// TwinCAT 3 PLC project Struckig
// Title: Struckig
// Company: Stefan Besler
// Author: Stefan Besler and contributers
// ProjectVersion: 0.19.4.0
// Description: Full port of pantor ruckig library (Community version) to IEC 61131-3 Structured Text. Online Trajectory Generation. Real-time. Time-optimal. Jerk-constrained.
// ProgramVersion: 3.1.4026.18
// project tree:
//   / Constants.TcGVL, ParameterList.TcGVL
//   Struckig/Block/ BlockInterval.TcDUT, Block.TcDUT
//   Struckig/BrakeProfile/ BrakeProfile.TcPOU
//   Struckig/ Integrate.TcPOU, IOtg.TcIO, Otg1.TcPOU, Otg.TcPOU
//   Struckig/Math/ BubbleSortLreal.TcPOU, Ceil.TcPOU, Clamp.TcPOU, Fmod.TcPOU, IsNaN.TcPOU, IsInfinity.TcPOU, LrealBits.TcPOU, LrealFromBits.TcPOU, Power.TcPOU, Power2.TcPOU, Cbrt.TcPOU, Roots.TcPOU
//   Struckig/Position/ PositionFirstOrderStep1.TcPOU, PositionFirstOrderStep2.TcPOU, PositionThirdOrderStep1.TcPOU, PositionSecondOrderStep1.TcPOU, PositionThirdOrderStep2.TcPOU, PositionSecondOrderStep2.TcPOU
//   Struckig/Profile/ ProfileDesc.TcPOU
//   Struckig/Profile/_DataTypes/ ProfileBound.TcDUT, ProfileDirection.TcDUT, ProfileControlSigns.TcDUT, ReachedLimits.TcDUT
//   Struckig/Velocity/ VelocitySecondOrderStep2.TcPOU, VelocityThirdOrderStep1.TcPOU, VelocitySecondOrderStep1.TcPOU, VelocityThirdOrderStep2.TcPOU
//   Struckig/_DataTypes/ ControlInterfaceType.TcDUT, DiscretizationType.TcDUT, SynchronizationType.TcDUT, TrajectoryErrorCode.TcDUT, TrajectoryState.TcDUT

// ---- Struckig/Block/BlockInterval.TcDUT
// Struckig
// Copyright (C) 2022 Stefan Besler

// This program is free software: you can redistribute it and/or modify
// it under the terms of the GNU General Public License as published by
// the Free Software Foundation, either version 3 of the License, or
// (at your option) any later version.

// This program is distributed in the hope that it will be useful,
// but WITHOUT ANY WARRANTY; without even the implied warranty of
// MERCHANTABILITY or FITNESS FOR A PARTICULAR PURPOSE.  See the
// GNU General Public License for more details.
//
// You should have received a copy of the GNU General Public License
// along with THIS PROGRAM.  IF NOT, see <http://www.gnu.org/licenses/>.
/// Which times are possible for synchronization?
TYPE INTERNAL BlockInterval :
STRUCT
  IsUsed : BOOL;
  Left, Right : LREAL;
  Profile : ProfileDesc;
END_STRUCT
END_TYPE

// ---- Struckig/Block/Block.TcDUT
// Struckig
// Copyright (C) 2022 Stefan Besler

// This program is free software: you can redistribute it and/or modify
// it under the terms of the GNU General Public License as published by
// the Free Software Foundation, either version 3 of the License, or
// (at your option) any later version.

// This program is distributed in the hope that it will be useful,
// but WITHOUT ANY WARRANTY; without even the implied warranty of
// MERCHANTABILITY or FITNESS FOR A PARTICULAR PURPOSE.  See the
// GNU General Public License for more details.
//
// You should have received a copy of the GNU General Public License
// along with THIS PROGRAM.  IF NOT, see <http://www.gnu.org/licenses/>.
TYPE INTERNAL Block :
STRUCT
  Pmin : ProfileDesc; // Save min Profile so that it doesn't need to be recalculated in Step2
  Tmin : LREAL; // [s]
  A, B : BlockInterval; // Max. 2 intervals can be blocked: called a and b with corresponding profiles, order does not matter  
END_STRUCT
END_TYPE

// ---- Struckig/Profile/_DataTypes/ProfileBound.TcDUT
// Struckig
// Copyright (C) 2022 Stefan Besler

// This program is free software: you can redistribute it and/or modify
// it under the terms of the GNU General Public License as published by
// the Free Software Foundation, either version 3 of the License, or
// (at your option) any later version.

// This program is distributed in the hope that it will be useful,
// but WITHOUT ANY WARRANTY; without even the implied warranty of
// MERCHANTABILITY or FITNESS FOR A PARTICULAR PURPOSE.  See the
// GNU General Public License for more details.
//
// You should have received a copy of the GNU General Public License
// along with THIS PROGRAM.  IF NOT, see <http://www.gnu.org/licenses/>.
{attribute 'conditionalshow'}
/// Positional envelope of a single-DoF profile.
/// The structure stores minimum/maximum position and the corresponding
/// times where these extrema occur along the generated trajectory.
///
/// It is returned by profile-bound checks to answer questions such as:
/// "What is the furthest negative/positive excursion and when does it happen?"
TYPE ProfileBound :
STRUCT
  Minimum, Maximum : LREAL; //< Extreme positions reached by the profile.
  Tmin, Tmax : LREAL;  //< Times at which `Minimum` and `Maximum` are reached.
END_STRUCT
END_TYPE

// ---- Struckig/Profile/_DataTypes/ProfileDirection.TcDUT
// Struckig
// Copyright (C) 2022 Stefan Besler

// This program is free software: you can redistribute it and/or modify
// it under the terms of the GNU General Public License as published by
// the Free Software Foundation, either version 3 of the License, or
// (at your option) any later version.

// This program is distributed in the hope that it will be useful,
// but WITHOUT ANY WARRANTY; without even the implied warranty of
// MERCHANTABILITY or FITNESS FOR A PARTICULAR PURPOSE.  See the
// GNU General Public License for more details.
//
// You should have received a copy of the GNU General Public License
// along with THIS PROGRAM.  IF NOT, see <http://www.gnu.org/licenses/>.
{attribute 'qualified_only'}
{attribute 'strict'}
TYPE INTERNAL ProfileDirection :
(
  Up,
  Down
);
END_TYPE

// ---- Struckig/Profile/_DataTypes/ProfileControlSigns.TcDUT
// Struckig
// Copyright (C) 2022 Stefan Besler

// This program is free software: you can redistribute it and/or modify
// it under the terms of the GNU General Public License as published by
// the Free Software Foundation, either version 3 of the License, or
// (at your option) any later version.

// This program is distributed in the hope that it will be useful,
// but WITHOUT ANY WARRANTY; without even the implied warranty of
// MERCHANTABILITY or FITNESS FOR A PARTICULAR PURPOSE.  See the
// GNU General Public License for more details.
//
// You should have received a copy of the GNU General Public License
// along with THIS PROGRAM.  IF NOT, see <http://www.gnu.org/licenses/>.
{attribute 'qualified_only'}
{attribute 'strict'}
TYPE INTERNAL ProfileControlSigns :
(
  Uddu,
  Udud 
);
END_TYPE

// ---- Struckig/Profile/_DataTypes/ReachedLimits.TcDUT
// Struckig
// Copyright (C) 2022 Stefan Besler

// This program is free software: you can redistribute it and/or modify
// it under the terms of the GNU General Public License as published by
// the Free Software Foundation, either version 3 of the License, or
// (at your option) any later version.

// This program is distributed in the hope that it will be useful,
// but WITHOUT ANY WARRANTY; without even the implied warranty of
// MERCHANTABILITY or FITNESS FOR A PARTICULAR PURPOSE.  See the
// GNU General Public License for more details.
//
// You should have received a copy of the GNU General Public License
// along with THIS PROGRAM.  IF NOT, see <http://www.gnu.org/licenses/>.
{attribute 'qualified_only'}
{attribute 'strict'}
TYPE INTERNAL ReachedLimits :
(
  Acc0Acc1Vel,
  Vel, 
  Acc0,
  Acc1,
  Acc0Acc1,
  Acc0Vel,
  Acc1Vel,
  None
);
END_TYPE

// ---- Struckig/_DataTypes/ControlInterfaceType.TcDUT
// Struckig
// Copyright (C) 2022 Stefan Besler

// This program is free software: you can redistribute it and/or modify
// it under the terms of the GNU General Public License as published by
// the Free Software Foundation, either version 3 of the License, or
// (at your option) any later version.

// This program is distributed in the hope that it will be useful,
// but WITHOUT ANY WARRANTY; without even the implied warranty of
// MERCHANTABILITY or FITNESS FOR A PARTICULAR PURPOSE.  See the
// GNU General Public License for more details.
//
// You should have received a copy of the GNU General Public License
// along with THIS PROGRAM.  IF NOT, see <http://www.gnu.org/licenses/>.
{attribute 'qualified_only'}
{attribute 'strict'}
/// Defines the controlled state variables for trajectory generation.
/// The selected mode changes which boundary values and limits are interpreted
/// during validation and profile generation.
TYPE ControlInterfaceType :
(
  Undefined, //< Use global/default configuration.
  Position, //< Full control over position, velocity, and acceleration.
  Velocity //< Controls only velocity and acceleration states.
);
END_TYPE

// ---- Struckig/_DataTypes/DiscretizationType.TcDUT
// Struckig
// Copyright (C) 2022 Stefan Besler

// This program is free software: you can redistribute it and/or modify
// it under the terms of the GNU General Public License as published by
// the Free Software Foundation, either version 3 of the License, or
// (at your option) any later version.

// This program is distributed in the hope that it will be useful,
// but WITHOUT ANY WARRANTY; without even the implied warranty of
// MERCHANTABILITY or FITNESS FOR A PARTICULAR PURPOSE.  See the
// GNU General Public License for more details.
//
// You should have received a copy of the GNU General Public License
// along with THIS PROGRAM.  IF NOT, see <http://www.gnu.org/licenses/>.
{attribute 'qualified_only'}
{attribute 'strict'}
/// Defines whether synchronized trajectory duration is continuous or cycle-discrete.
TYPE DiscretizationType :
(
  Continuous, //< Every synchronization duration is allowed.
  Discrete //< Synchronization duration must be a multiple of cycle time.
);
END_TYPE

// ---- Struckig/_DataTypes/SynchronizationType.TcDUT
// Struckig
// Copyright (C) 2022 Stefan Besler

// This program is free software: you can redistribute it and/or modify
// it under the terms of the GNU General Public License as published by
// the Free Software Foundation, either version 3 of the License, or
// (at your option) any later version.

// This program is distributed in the hope that it will be useful,
// but WITHOUT ANY WARRANTY; without even the implied warranty of
// MERCHANTABILITY or FITNESS FOR A PARTICULAR PURPOSE.  See the
// GNU General Public License for more details.
//
// You should have received a copy of the GNU General Public License
// along with THIS PROGRAM.  IF NOT, see <http://www.gnu.org/licenses/>.
{attribute 'qualified_only'}
{attribute 'strict'}
/// Defines how multiple DoFs are synchronized to a common trajectory timing.
/// This setting is evaluated together with per-axis overrides (`PerDofSynchronization`)
/// in [Otg](xref:Struckig.Otg).
TYPE SynchronizationType :
(
  Undefined, //< Use global/default configuration.
  TimeSync, //< Always synchronize the DoFs to reach the target at the same time (Default)
  TimeIfNecessarySync, //< Synchronize only when necessary (e.g. for non-zero target velocity or acceleration)
  Phase,  //< Phase synchronize the DoFs when this is possible, else fallback to "Time" strategy. Phase synchronization will result a straight-line trajectory
    // PhaseOnly, //< Always phase synchronize the DoFs (even when this is not time-optimal), else returns "ErrorNoPhaseSynchronization". Ruckig will then guarantee a straight-line trajectory
  None //< Calculate every DoF independently
);
END_TYPE

// ---- Struckig/_DataTypes/TrajectoryErrorCode.TcDUT
// Struckig
// Copyright (C) 2022 Stefan Besler

// This program is free software: you can redistribute it and/or modify
// it under the terms of the GNU General Public License as published by
// the Free Software Foundation, either version 3 of the License, or
// (at your option) any later version.

// This program is distributed in the hope that it will be useful,
// but WITHOUT ANY WARRANTY; without even the implied warranty of
// MERCHANTABILITY or FITNESS FOR A PARTICULAR PURPOSE.  See the
// GNU General Public License for more details.
//
// You should have received a copy of the GNU General Public License
// along with THIS PROGRAM.  IF NOT, see <http://www.gnu.org/licenses/>.
{attribute 'qualified_only'}
/// Error codes reported by the trajectory generator.
/// Returned by [ErrorCode](xref:Struckig.IOtg#ErrorCode) and explained by
/// [ErrorMessage](xref:Struckig.IOtg#ErrorMessage).
TYPE TrajectoryErrorCode :
(
  Undefined := 0, //< No error.
  InvalidInput, //< Error in the input parameter
  SynchronizationFailed, //< No valid synchronized profile was found.
  CalculateStep1Failed, //< Profile search in step 1 failed.
  ZeroLimitsConflict, //< Conflicting zero limits prevent profile generation.
  ZeroLimitsConflictInSynchronization //< Zero-limit conflict during multi-DoF synchronization.
);
END_TYPE

// ---- Struckig/_DataTypes/TrajectoryState.TcDUT
// Struckig
// Copyright (C) 2022 Stefan Besler

// This program is free software: you can redistribute it and/or modify
// it under the terms of the GNU General Public License as published by
// the Free Software Foundation, either version 3 of the License, or
// (at your option) any later version.

// This program is distributed in the hope that it will be useful,
// but WITHOUT ANY WARRANTY; without even the implied warranty of
// MERCHANTABILITY or FITNESS FOR A PARTICULAR PURPOSE.  See the
// GNU General Public License for more details.
//
// You should have received a copy of the GNU General Public License
// along with THIS PROGRAM.  IF NOT, see <http://www.gnu.org/licenses/>.
{attribute 'qualified_only'}
{attribute 'strict'}
/// Runtime state of the trajectory generator.
TYPE TrajectoryState :
(
  Undefined, //< State has not been initialized yet.
  
  /// The trajectory has reached its final position. For trajectories with a target velocity or/and a target acceleration
  /// there will still be movement.
  Idle,
  
  /// The trajectory is calculated normally
  Busy,
  
  /// An error occured, use [ErrorCode](xref:Struckig.IOtg#ErrorCode) and [ErrorMessage](xref:Struckig.IOtg#ErrorMessage) to get more
  /// information about the error.
  Error
);
END_TYPE

// ---- Constants.TcGVL
// Struckig
// Copyright (C) 2022 Stefan Besler

// This program is free software: you can redistribute it and/or modify
// it under the terms of the GNU General Public License as published by
// the Free Software Foundation, either version 3 of the License, or
// (at your option) any later version.

// This program is distributed in the hope that it will be useful,
// but WITHOUT ANY WARRANTY; without even the implied warranty of
// MERCHANTABILITY or FITNESS FOR A PARTICULAR PURPOSE.  See the
// GNU General Public License for more details.
//
// You should have received a copy of the GNU General Public License
// along with THIS PROGRAM.  IF NOT, see <http://www.gnu.org/licenses/>.
{attribute 'qualified_only'}
{attribute 'hide'}
VAR_GLOBAL CONSTANT
  BrakeEpsilon : LREAL := 2.2E-14;
  DoubleEpsilon : LREAL := 2.2204460492503131E-016; // smallest such that 1.0+Constants.DoubleEpsilon != 1.0
  Epsilon : LREAL := 1E-8;
  Epsilon16 : LREAL := 16 * 2.2204460492503131E-016;
  EpsilonColinear : LREAL := 1E-7;
  Infinity : LREAL := 1.7976931348623157E+308;  
  Tolerance : LREAL := 1E-14;
  Cos120 : LREAL := -0.50;
  Sin120 : LREAL := 0.866025403784438646764;  
  Pi : LREAL := 3.14159265358979323846;
  Minimum : LREAL := 1.17549435082E-38;  // used for validating input
  
  VelocityEpsilon : LREAL := 1E-12;
  AccelerationEpsilon : LREAL := 1E-12;
  JerkEpsilon : LREAL := 1E-12; 
  
  PositionPrecision : LREAL := 1E-8;
  VelocityPrecision : LREAL := 1E-8;
  AccelerationPrecision : LREAL := 1E-10;
  TimePrecision : LREAL := 1E-12;  
  
  Tmax : LREAL := 1E12;
END_VAR

// ---- ParameterList.TcGVL
// Struckig
// Copyright (C) 2022 Stefan Besler

// This program is free software: you can redistribute it and/or modify
// it under the terms of the GNU General Public License as published by
// the Free Software Foundation, either version 3 of the License, or
// (at your option) any later version.

// This program is distributed in the hope that it will be useful,
// but WITHOUT ANY WARRANTY; without even the implied warranty of
// MERCHANTABILITY or FITNESS FOR A PARTICULAR PURPOSE.  See the
// GNU General Public License for more details.
//
// You should have received a copy of the GNU General Public License
// along with THIS PROGRAM.  IF NOT, see <http://www.gnu.org/licenses/>.
{attribute 'qualified_only'}
/// Global configuration constants for Struckig.
/// These values define library limits and algorithm defaults that are
/// referenced by trajectory generation and numerical helper routines.
VAR_GLOBAL CONSTANT
  MaxDoFs : INT := 7; //< Maximum number of degrees of freedom supported by `Otg`.
  MaxIterations : BYTE := 127; //< Maximum iterations when [shrinking an interval](xref:Struckig.Roots#ShrinkInterval)
  NumericalRobust : BOOL := TRUE; //< Enables additional guards for numerically robust calculations.
  
  /// Default initial value for Otg.SmoothBrake / Otg1.SmoothBrake
  /// If enabled, braking profiles prefer smooth acceleration transitions.
  SmoothBrake : BOOL := FALSE;
END_VAR

// ---- Struckig/IOtg.TcIO
// Struckig
// Copyright (C) 2022 Stefan Besler

// This program is free software: you can redistribute it and/or modify
// it under the terms of the GNU General Public License as published by
// the Free Software Foundation, either version 3 of the License, or
// (at your option) any later version.

// This program is distributed in the hope that it will be useful,
// but WITHOUT ANY WARRANTY; without even the implied warranty of
// MERCHANTABILITY or FITNESS FOR A PARTICULAR PURPOSE.  See the
// GNU General Public License for more details.
//
// You should have received a copy of the GNU General Public License
// along with THIS PROGRAM.  IF NOT, see <http://www.gnu.org/licenses/>.
/// Public interface for Struckig online trajectory generators.
/// The interface unifies access to both [Otg](xref:Struckig.Otg) (multi-DoF)
/// and [Otg1](xref:Struckig.Otg1) (single-DoF wrapper), so user code can
/// switch implementation without changing call sites.
///
/// A typical pattern is:
/// 1. Call `Cyclic` each PLC cycle.
/// 2. Monitor `State`.
/// 3. Read command setpoints from the concrete implementation outputs.
/// 4. Use `Reset` and `ValidateInput` for robust operation.
INTERFACE IOtg

/// \copydoc Struckig.Otg#AtTime
{attribute 'conditionalshow'}
METHOD AtTime
VAR_INPUT
  t : LREAL;
  new_position : POINTER TO LREAL;
  new_velocity : POINTER TO LREAL;
  new_acceleration : POINTER TO LREAL;
  new_jerk : POINTER TO LREAL;  
  new_section : POINTER TO INT;
END_VAR
END_METHOD

/// \copydoc Struckig.Otg#AtTime1
{attribute 'conditionalshow'}
METHOD AtTime1
VAR_INPUT
  t : LREAL;
  new_position : REFERENCE TO LREAL;
  new_velocity : REFERENCE TO LREAL;
  new_acceleration : REFERENCE TO LREAL;
  new_jerk : REFERENCE TO LREAL;
END_VAR
END_METHOD

/// \copydoc Struckig.Otg#Cyclic
METHOD Cyclic
VAR_INPUT
END_VAR
END_METHOD

/// \copydoc Struckig.Otg#Duration
PROPERTY Duration : LREAL
GET
END_GET
END_PROPERTY

/// \copydoc Struckig.Otg#ErrorCode
METHOD ErrorCode : TrajectoryErrorCode
VAR_INPUT
END_VAR
END_METHOD

/// \copydoc Struckig.Otg#ErrorMessage
METHOD ErrorMessage : STRING(255)
VAR_INPUT
END_VAR
END_METHOD

/// \copydoc Struckig.Otg#PassOutputToInput
METHOD PassOutputToInput
VAR_INPUT
END_VAR
END_METHOD

/// \copydoc Struckig.Otg#Reset
METHOD Reset
VAR_INPUT
END_VAR
END_METHOD

/// \copydoc Struckig.Otg#State
PROPERTY State : TrajectoryState
GET
END_GET
END_PROPERTY

/// \copydoc Struckig.Otg#ValidateInput
{attribute 'conditionalshow'}
METHOD ValidateInput : BOOL
VAR_INPUT
  checkCurrentStateWithinLimits : BOOL;
  checkTargetStateWithinLimits : BOOL;
END_VAR
END_METHOD

END_INTERFACE

// ---- Struckig/Otg.TcPOU
// Struckig
// Copyright (C) 2022 Stefan Besler

// This program is free software: you can redistribute it and/or modify
// it under the terms of the GNU General Public License as published by
// the Free Software Foundation, either version 3 of the License, or
// (at your option) any later version.

// This program is distributed in the hope that it will be useful,
// but WITHOUT ANY WARRANTY; without even the implied warranty of
// MERCHANTABILITY or FITNESS FOR A PARTICULAR PURPOSE.  See the
// GNU General Public License for more details.
//
// You should have received a copy of the GNU General Public License
// along with THIS PROGRAM.  IF NOT, see <http://www.gnu.org/licenses/>.
{attribute 'conditionalshow_all_locals'}
/// Online trajectory generator for multiple DoFs.
/// Call the function block cyclically to generate smooth, time-optimal motion
/// under position, velocity, acceleration, and jerk limits.
///
/// Typical cycle:
/// 1. Set current state, target state, and limits.
/// 2. Call the function block every PLC cycle.
/// 3. Use `NewPosition`, `NewVelocity`, `NewAcceleration`, and `NewJerk` as command values.
/// 4. Optionally call [PassOutputToInput](xref:Struckig.Otg#PassOutputToInput) or enable
///    `EnableAutoPropagate` for state propagation.
///
/// ```st
/// otg(
///   CycleTime := 0.001,
///   Dofs := 2,
///   ControlInterface := ControlInterfaceType.Position,
///   Synchronization := SynchronizationType.TimeSync
/// );
///
/// IF otg.State = TrajectoryState.Busy THEN
///   Axis1.Setpoint := otg.NewPosition[0];
///   Axis2.Setpoint := otg.NewPosition[1];
/// END_IF
/// ```
FUNCTION_BLOCK Otg IMPLEMENTS IOtg
VAR_INPUT
  CycleTime : LREAL;
  Dofs : INT;
  Enabled : ARRAY[0..ParameterList.MaxDoFs] OF BOOL;  
  ControlInterface : ControlInterfaceType := ControlInterfaceType.Position; //< The default position interface controls the full kinematic state.
  Synchronization : SynchronizationType := SynchronizationType.TimeSync; //< Synchronization behavior of multiple DoFs
  PerDofControlInterface : ARRAY[0..ParameterList.MaxDoFs] OF ControlInterfaceType; //< Per-DoF control interface (overwrites global ControlInterface)
  PerDofSynchronization: ARRAY[0..ParameterList.MaxDoFs] OF SynchronizationType; //< Per-DoF synchronization (overwrites global Synchronization)
  Discretization : DiscretizationType; //< Whether the duration should be a discrete multiple of the control cycle (off by default)
  CurrentPosition, CurrentVelocity, CurrentAcceleration : ARRAY[0..ParameterList.MaxDoFs] OF LREAL; //< Current state
  TargetPosition, TargetVelocity, TargetAcceleration : ARRAY[0..ParameterList.MaxDoFs] OF LREAL; //< Target state
  MaxVelocity : ARRAY[0..ParameterList.MaxDoFs] OF LREAL; //< Kinematic constraints
  MaxAcceleration : ARRAY[0..ParameterList.MaxDoFs] OF LREAL; //< Kinematic constraints, defaults to Infinity (Struckig.Constants.Infinity)
  MaxJerk : ARRAY[0..ParameterList.MaxDoFs] OF LREAL; //< Kinematic constraints, defaults to Infinity (Struckig.Constants.Infinity)
  MinVelocity, MinAcceleration : ARRAY[0..ParameterList.MaxDoFs] OF LREAL; //< Optional kindematic constraints
  MinDuration : LREAL := 0; //< Optional minimum duration of a trajectory. This is only considered if the Synchronization type is not none
  EnableAutoPropagate : BOOL; //< If set to true, PassOutputToInput is automatically called internally after calling the function block's body
  SmoothBrake : BOOL := ParameterList.SmoothBrake; //< Initialized from ParameterList; override per instance if needed
END_VAR
VAR_OUTPUT
  NewPosition, NewVelocity, NewAcceleration, NewJerk : ARRAY[0..ParameterList.MaxDoFs] OF LREAL;
  NewCalculation : BOOL; //< Was a new trajectory calculation performed in the last cycle?
  CurrentTime : LREAL; //< Time elapsed on the current trajectory in seconds.
END_VAR
VAR
  _duration : LREAL;
  _state : TrajectoryState;  
  _inputInitialized : BOOL := FALSE;
  _newSection : INT; //< not used in Struckig, ruckig pro feature
  _blocks : ARRAY[0..ParameterList.MaxDoFs] OF Block;  
  _profiles : ARRAY[0..ParameterList.MaxDoFs] OF ProfileDesc;
  _independentMinDurations : ARRAY[0..ParameterList.MaxDoFs] OF LREAL;
  
  _positionThirdOrderStep1 : PositionThirdOrderStep1;
  _positionThirdOrderStep2 : PositionThirdOrderStep2;
  _velocityThirdOrderStep1 : VelocityThirdOrderStep1;
  _velocityThirdOrderStep2 : VelocityThirdOrderStep2;
  
  _positionSecondOrderStep1 : PositionSecondOrderStep1;
  _positionSecondOrderStep2 : PositionSecondOrderStep2;
  _velocitySecondOrderStep1 : VelocitySecondOrderStep1;
  _velocitySecondOrderStep2 : VelocitySecondOrderStep2;
  
  _positionFirstOrderStep1 : PositionFirstOrderStep1;
  _positionFirstOrderStep2 : PositionFirstOrderStep2;  
  
  _inp_min_velocity, _inp_min_acceleration : ARRAY[0..ParameterList.MaxDoFs] OF LREAL;
  _inp_per_dof_control_interface : ARRAY[0..ParameterList.MaxDoFs] OF ControlInterfaceType; //< Per-DoF control interface
  _inp_per_dof_synchronization : ARRAY[0..ParameterList.MaxDoFs] OF SynchronizationType; //< Per-DoF synchronization
  
  _dofs, _dofsEnd : INT;
  _enabled : ARRAY[0..ParameterList.MaxDoFs] OF BOOL;  
  _controlInterface : ControlInterfaceType := ControlInterfaceType.Position; //< The default position interface controls the full kinematic state.
  _synchronization : SynchronizationType := SynchronizationType.TimeSync; //< Synchronization behavior of multiple DoFs
  _perDofControlInterface : ARRAY[0..ParameterList.MaxDoFs] OF ControlInterfaceType; //< Per-DoF control interface
  _perDofSynchronization: ARRAY[0..ParameterList.MaxDoFs] OF SynchronizationType; //< Per-DoF synchronization
  _discretization : DiscretizationType; //< Whether the duration should be a discrete multiple of the control cycle (off by default)
  _currentPosition, _currentVelocity, _currentAcceleration : ARRAY[0..ParameterList.MaxDoFs] OF LREAL; //< Current state
  _targetPosition, _targetVelocity, _targetAcceleration : ARRAY[0..ParameterList.MaxDoFs] OF LREAL; //< Target state
  _maxVelocity, _maxAcceleration, _maxJerk : ARRAY[0..ParameterList.MaxDoFs] OF LREAL; //< Kinematic constraints
  _new_phase_control : ARRAY[0..ParameterList.MaxDoFs] OF LREAL;
  _minVelocity, _minAcceleration : ARRAY[0..ParameterList.MaxDoFs] OF LREAL; //< Optional kindematic constraints
  _minDuration : LREAL := 0; //< Optional minimum duration of a trajectory. This is only considered if the Synchronization type is not none
  _smoothBrake : BOOL;
  _dt : LREAL; //< Time step between updates (cycle time) in [s]
  _errorId : INT;
  _errorMessage : STRING(255);
END_VAR

NewCalculation := FALSE;
SetBusy(TRUE);

IF NOT _inputInitialized OR_ELSE HasChanged() 
THEN
  _dofsEnd := Dofs - 1; // for looping

  Calculate();
  IF State = TrajectoryState.Error THEN
    RETURN;
  END_IF

  // Store the desired state to check for potential changes
  _dofs := Dofs;
  _enabled := Enabled;
  _controlInterface := ControlInterface;
  _synchronization := Synchronization;
  _discretization := Discretization;
  _currentPosition := CurrentPosition;
  _currentVelocity := CurrentVelocity;
  _currentAcceleration := CurrentAcceleration;
  _targetPosition := TargetPosition;
  _targetVelocity := TargetVelocity;
  _targetAcceleration := TargetAcceleration;
  _maxVelocity := MaxVelocity;
  _maxAcceleration := MaxAcceleration;
  _maxJerk := MaxJerk;
  _minVelocity := MinVelocity;
  _minAcceleration := MinAcceleration;
  _minDuration := MinDuration;
  _smoothBrake := SmoothBrake;
  _perDofControlInterface := PerDofControlInterface;
  _perDofSynchronization := PerDofSynchronization;
  _dt := CycleTime;
  _inputInitialized := TRUE;
  CurrentTime := 0.0;
  NewCalculation := TRUE;  
END_IF

CurrentTime := CurrentTime + _dt;
AtTime(CurrentTime, ADR(NewPosition), ADR(NewVelocity), ADR(NewAcceleration), ADR(NewJerk), ADR(_newSection));

_currentPosition := NewPosition;
_currentVelocity := NewVelocity;
_currentAcceleration := NewAcceleration;

IF CurrentTime > _duration THEN
  _state := TrajectoryState.Idle;
END_IF

IF EnableAutoPropagate
THEN
  PassOutputToInput();
END_IF

METHOD PROTECTED AbortErrorId
VAR_INPUT
  errorId : INT;
END_VAR
VAR_IN_OUT CONSTANT  
  message : STRING;
END_VAR
_state := TrajectoryState.Error;
_errorMessage := message;
_errorId := errorId;
END_METHOD

/// Gets the kinematic state at absolute trajectory time `t`.
/// This method evaluates the active profile sections and returns position, velocity,
/// acceleration, and jerk for each configured DoF.
///
/// For `t >= Duration`, the final state is extended with constant acceleration behavior.
/// For single-axis access without vector pointers, see [AtTime1](xref:Struckig.Otg#AtTime1).
{attribute 'conditionalshow'}
METHOD AtTime
VAR_INPUT
  t : LREAL;
  new_position : POINTER TO LREAL;
  new_velocity : POINTER TO LREAL;
  new_acceleration : POINTER TO LREAL;
  new_jerk : POINTER TO LREAL;
  new_section : POINTER TO INT;
END_VAR
VAR
  dof : INT;
  p : REFERENCE TO ProfileDesc;
  t_diff : LREAL;
  index : INT;
END_VAR
IF (t >= Duration) THEN
  // Keep constant acceleration
  //new_section := 1;
  FOR dof:=0 TO _dofsEnd DO
    Integrate(t - (_profiles[dof].Brake.Duration + _profiles[dof].t_sum[6]), _profiles[dof].p[7], _profiles[dof].v[7], _profiles[dof].a[7], 0, p:=new_position[dof], v:=new_velocity[dof], a:=new_acceleration[dof]);
    new_jerk[dof] := 0;
  END_FOR
  RETURN;
END_IF

//new_section := 0;
FOR dof:=0 TO _dofsEnd DO
  p REF= _profiles[dof];

  t_diff := t;
  
  // Brake pre-trajectory
  IF (p.Brake.Duration > 0) THEN
    IF (t_diff < p.Brake.Duration) THEN
      IF t_diff < p.Brake.t[0] THEN
        index := 0;
      ELSIF t_diff < p.Brake.t[0] + p.Brake.t[1] THEN
        index := 1;
        t_diff := t_diff - p.Brake.t[0];
      ELSE
        index := 2;
        t_diff := t_diff - p.Brake.t[0] - p.Brake.t[1];
      END_IF

      Integrate(t_diff, p.Brake.p[index], p.Brake.v[index], p.Brake.a[index], p.Brake.j[index], p:=new_position[dof], v:=new_velocity[dof], a:=new_acceleration[dof]);
      new_jerk[dof] := p.Brake.j[index];
      CONTINUE;
    ELSE
      t_diff := t_diff - p.Brake.Duration;
    END_IF
  END_IF
  
// Accel post-trajectory
// if (new_section == profiles.size() - 1 && p.accel.duration > 0) {
//     if (t_diff_dof > p.t_sum[6]) {
//         const size_t index = (t_diff_dof < p.accel.t[0]) ? 1 : 0;
//         if (index > 0) {
//             t_diff_dof -= p.accel.t[index - 1];
//         }

//         std::tie(new_position[dof], new_velocity[dof], new_acceleration[dof]) = integrate(t_diff_dof, p.accel.p[index], p.accel.v[index], p.accel.a[index], p.accel.j[index]);
//         continue;
//     }
// }

  // Non-time synchronization
  IF (t_diff >= p.t_sum[6]) THEN
    // Keep constant acceleration
    Integrate(t_diff - p.t_sum[6], p.p[7], p.v[7], p.a[7], 0, p:=new_position[dof], v:=new_velocity[dof], a:=new_acceleration[dof]);
    new_jerk[dof] := 0;    
    CONTINUE;
  END_IF

  FOR index:=0 TO 6 DO
    IF p.t_sum[index] > t_diff
    THEN
      EXIT;
    END_IF
	END_FOR
  
  IF (index > 0) THEN
    t_diff := t_diff - p.t_sum[index - 1];
  END_IF

  Integrate(t_diff, p.p[index], p.v[index], p.a[index], p.j[index], p:=new_position[dof], v:=new_velocity[dof], a:=new_acceleration[dof]);
  new_jerk[dof] := p.j[index];      
END_FOR
END_METHOD

/// Get the kinematic state and current section at a given time without vectors for a single DoF.
/// Using this method is only allowed for DoF = 1, for higher degrees of freedom use
/// [AtTime](xref:Struckig.Otg#AtTime). Using this method for DoF > 0 will not yield any result
{attribute 'conditionalshow'}
METHOD AtTime1
VAR_INPUT
  t : LREAL;
  new_position : REFERENCE TO LREAL;
  new_velocity : REFERENCE TO LREAL;
  new_acceleration : REFERENCE TO LREAL;
  new_jerk : REFERENCE TO LREAL;  
END_VAR
IF _dofs = 1
THEN
  AtTime(t, ADR(new_position), ADR(new_velocity), ADR(new_acceleration), ADR(new_jerk), 0);
END_IF
END_METHOD

METHOD PRIVATE Calculate
VAR_INST
  dof, i : INT;
  p, p_limiting : REFERENCE TO ProfileDesc;
  found_profile : BOOL;
  limiting_dof : INT := -1; // The DoF that doesn't need step 2
  discrete_duration, found_synchronization, found_time_synchronization : BOOL;
  t_profile : LREAL;
  noneSynchronizationCount, phaseSychronizations, phaseOrNoneSychronizationCount : INT;
  has_zero_limits : BOOL;
  _smooth_profile : ProfileDesc;
  _smooth_block : Block;
  _smooth_found : BOOL;
END_VAR
SetBusy(TRUE);
IF NOT ValidateInputOrAbort(checkCurrentStateWithinLimits:=FALSE, checkTargetStateWithinLimits:=TRUE)
THEN
  RETURN;
END_IF

FOR dof:=0 TO _dofsEnd
DO
  p REF=_profiles[dof];
  
  _inp_min_velocity[dof] := SEL(ABS(MinVelocity[dof]) < Constants.Epsilon, MinVelocity[dof], -MaxVelocity[dof]);
  _inp_min_acceleration[dof] := SEL(ABS(MinAcceleration[dof]) < Constants.Epsilon, MinAcceleration[dof], -MaxAcceleration[dof]);
  _inp_per_dof_control_interface[dof] := SEL(PerDofControlInterface[dof] = ControlInterfaceType.Undefined, PerDofControlInterface[dof], ControlInterface);
  _inp_per_dof_synchronization[dof] := SEL(PerDofSynchronization[dof] = SynchronizationType.Undefined, PerDofSynchronization[dof], Synchronization); 
  
  IF NOT Enabled[dof]
  THEN
    p.p[7] := CurrentPosition[dof];
    p.v[7] := CurrentVelocity[dof];
    p.a[7] := CurrentAcceleration[dof];    
    p.t_sum[6] := 0.0;
    _blocks[dof].Tmin := 0.0;
    _blocks[dof].A.IsUsed := FALSE;
    _blocks[dof].B.IsUsed := FALSE;    
    CONTINUE;
	END_IF
  
  CASE _inp_per_dof_control_interface[dof]
  OF
    ControlInterfaceType.Position:
    
      IF NOT IsInfinity(MaxJerk[dof])
      THEN
        p.Brake.PositionBrakeTrajectory(CurrentVelocity[dof], CurrentAcceleration[dof], MaxVelocity[dof], _inp_min_velocity[dof], MaxAcceleration[dof], _inp_min_acceleration[dof], MaxJerk[dof], SmoothBrake := SmoothBrake);
      ELSIF NOT IsInfinity(MaxAcceleration[dof])
      THEN
        p.Brake.SecondOrderPositionBrakeTrajectory(CurrentVelocity[dof], MaxVelocity[dof], _inp_min_velocity[dof], MaxAcceleration[dof], _inp_min_acceleration[dof]);
      END_IF    

      p.SetBoundaryPosition(CurrentPosition[dof], CurrentVelocity[dof], CurrentAcceleration[dof], TargetPosition[dof], TargetVelocity[dof], TargetAcceleration[dof]);

    ControlInterfaceType.Velocity:
      IF NOT IsInfinity(MaxJerk[dof])
      THEN    
        p.Brake.VelocityBrakeTrajectory(CurrentVelocity[dof], CurrentAcceleration[dof], MaxAcceleration[dof], _inp_min_acceleration[dof], MaxJerk[dof]);
      ELSIF NOT IsInfinity(MaxAcceleration[dof])
      THEN
        p.Brake.SecondOrderVelocityBrakeTrajectory();        
      END_IF
      
      p.SetBoundaryVelocity(CurrentPosition[dof], CurrentVelocity[dof], CurrentAcceleration[dof], TargetVelocity[dof], TargetAcceleration[dof]);      
	END_CASE
  
  IF NOT IsInfinity(MaxJerk[dof])
  THEN
    p.Brake.Finalize(p.p[0], p.v[0], p.a[0]);
  ELSIF NOT IsInfinity(MaxAcceleration[dof])
  THEN
    p.Brake.FinalizeSecondOrder(p.p[0], p.v[0], p.a[0]);    
  END_IF

  CASE _inp_per_dof_control_interface[dof]
  OF
    ControlInterfaceType.Position:
      IF NOT IsInfinity(MaxJerk[dof])
      THEN
        _positionThirdOrderStep1.Set(p.p[0], p.v[0], p.a[0], p.pf, p.vf, p.af, MaxVelocity[dof], _inp_min_velocity[dof], MaxAcceleration[dof], _inp_min_acceleration[dof], MaxJerk[dof]);
        found_profile := _positionThirdOrderStep1.Get(p, _blocks[dof]);      
      ELSIF NOT IsInfinity(MaxAcceleration[dof])
      THEN
        _positionSecondOrderStep1.Set(p.p[0], p.v[0], p.pf, p.vf, MaxVelocity[dof], _inp_min_velocity[dof], MaxAcceleration[dof], _inp_min_acceleration[dof]);
        found_profile := _positionSecondOrderStep1.Get(p, _blocks[dof]);          
      ELSE
        _positionFirstOrderStep1.Set(p.p[0], p.pf, MaxVelocity[dof], _inp_min_velocity[dof]);
        found_profile := _positionFirstOrderStep1.Get(p, _blocks[dof]);          
      END_IF

    ControlInterfaceType.Velocity:
      IF NOT IsInfinity(MaxJerk[dof])
      THEN    
        _velocityThirdOrderStep1.Set(p.v[0], p.a[0], p.vf, p.af, MaxAcceleration[dof], _inp_min_acceleration[dof], MaxJerk[dof]);
        found_profile := _velocityThirdOrderStep1.Get(p, _blocks[dof]);
      ELSIF NOT IsInfinity(MaxAcceleration[dof])
      THEN
        _velocitySecondOrderStep1.Set(p.v[0], p.vf, MaxAcceleration[dof], _inp_min_acceleration[dof]);
        found_profile := _velocitySecondOrderStep1.Get(p, _blocks[dof]);    
      END_IF  
	END_CASE

  IF SmoothBrake
     AND_THEN _inp_per_dof_control_interface[dof] = ControlInterfaceType.Position
     AND_THEN NOT IsInfinity(MaxJerk[dof])
     AND_THEN p.Brake.Duration > 0
  THEN
    _smooth_profile := p;
    _smooth_block := _blocks[dof];
    _smooth_found := found_profile;

    p.Brake.PositionBrakeTrajectory(CurrentVelocity[dof], CurrentAcceleration[dof], MaxVelocity[dof], _inp_min_velocity[dof], MaxAcceleration[dof], _inp_min_acceleration[dof], MaxJerk[dof], SmoothBrake := FALSE);
    p.SetBoundaryPosition(CurrentPosition[dof], CurrentVelocity[dof], CurrentAcceleration[dof], TargetPosition[dof], TargetVelocity[dof], TargetAcceleration[dof]);
    p.Brake.Finalize(p.p[0], p.v[0], p.a[0]);
    _positionThirdOrderStep1.Set(p.p[0], p.v[0], p.a[0], p.pf, p.vf, p.af, MaxVelocity[dof], _inp_min_velocity[dof], MaxAcceleration[dof], _inp_min_acceleration[dof], MaxJerk[dof]);
    found_profile := _positionThirdOrderStep1.Get(p, _blocks[dof]);

    IF _smooth_found AND_THEN (NOT found_profile OR_ELSE _smooth_block.Tmin <= _blocks[dof].Tmin) THEN
      p := _smooth_profile;
      _blocks[dof] := _smooth_block;
      found_profile := TRUE;
    END_IF
  END_IF

  IF NOT found_profile
  THEN
    has_zero_limits := (MaxAcceleration[dof] = 0.0 OR_ELSE _inp_min_acceleration[dof] = 0.0 OR_ELSE MaxJerk[dof] = 0.0);
    IF has_zero_limits
    THEN
      AbortErrorId(TrajectoryErrorCode.ZeroLimitsConflict, '');
      RETURN;
    ELSE 
      AbortErrorId(TrajectoryErrorCode.CalculateStep1Failed, '');      
      RETURN;
    END_IF
	END_IF

  _independentMinDurations[dof] := _blocks[dof].Tmin;
END_FOR


discrete_duration := (Discretization = DiscretizationType.Discrete);

IF (dofs = 0 AND_THEN MinDuration <> 0 AND_THEN discrete_duration <> 0)
THEN 
  _duration := _blocks[0].Tmin;
  _profiles[0] := _blocks[0].Pmin;
  RETURN;
END_IF

found_synchronization := Synchronize(discrete_duration, MinDuration, _duration, limiting_dof);
IF NOT found_synchronization
THEN
  has_zero_limits := FALSE;
  FOR i:=0 TO _dofsEnd
  DO
    IF MaxAcceleration[dof] = 0.0 OR_ELSE _inp_min_acceleration[dof] = 0.0 OR_ELSE MaxJerk[dof] = 0.0
    THEN
      has_zero_limits := TRUE;
      EXIT;
    END_IF
  END_FOR
      
  IF has_zero_limits
  THEN
    AbortErrorId(TrajectoryErrorCode.ZeroLimitsConflictInSynchronization, '');
    RETURN;
  ELSE
    AbortErrorId(TrajectoryErrorCode.SynchronizationFailed, '');
    RETURN;    
	END_IF    
END_IF

// None Synchronization
FOR dof:=0 TO _dofsEnd
DO
  IF Enabled[dof] AND_THEN _inp_per_dof_synchronization[dof] = SynchronizationType.None
  THEN
    _profiles[dof] := _blocks[dof].Pmin;
    IF _blocks[dof].Tmin > Duration
    THEN
      _duration := _blocks[dof].Tmin;
      limiting_dof := dof;
    END_IF
  END_IF
END_FOR

IF (Duration = 0.0) THEN
  // Copy all profiles for end state
  FOR dof:=0 TO _dofsEnd
  DO
    _profiles[dof] := _blocks[dof].Pmin;
  END_FOR
  RETURN;
END_IF

noneSynchronizationCount := -1;
phaseSychronizations := -1;
phaseOrNoneSychronizationCount := -1;
FOR dof:=0 TO _dofsEnd DO 
  IF _inp_per_dof_synchronization[dof] = SynchronizationType.None
  THEN
    noneSynchronizationCount := noneSynchronizationCount + 1;
    phaseOrNoneSychronizationCount := phaseOrNoneSychronizationCount + 1;
  ELSIF _inp_per_dof_synchronization[dof] = SynchronizationType.Phase
  THEN
    phaseOrNoneSychronizationCount := phaseOrNoneSychronizationCount + 1;
    phaseSychronizations := phaseSychronizations + 1;
  END_IF
END_FOR

IF NOT discrete_duration AND_THEN noneSynchronizationCount = _dofsEnd
THEN
  RETURN;
END_IF

IF limiting_dof >= 0 AND_THEN phaseSychronizations >= 0 THEN
  p_limiting REF= _profiles[limiting_dof];
  IF IsInputCollinear(p_limiting.Direction, limiting_dof, _new_phase_control) THEN
    found_time_synchronization := TRUE;
    FOR dof:=0 TO _dofsEnd DO
      IF NOT Enabled[dof] OR_ELSE dof = limiting_dof OR_ELSE _inp_per_dof_synchronization[dof] <> SynchronizationType.Phase THEN
        CONTINUE;
      END_IF

      p REF= _profiles[dof];
      t_profile := Duration - p.Brake.Duration - p.Accel.Duration;

      p.t := p_limiting.t; // Copy timing information from limiting DoF
      p.ControlSigns := p_limiting.ControlSigns;

      CASE _inp_per_dof_control_interface[dof]
      OF
        ControlInterfaceType.Position:
          CASE p.ControlSigns
          OF
            ProfileControlSigns.Uddu:
            
              IF NOT IsInfinity(MaxJerk[dof])
              THEN
                IF NOT p.CheckWithTiming2(ProfileControlSigns.Uddu, ReachedLimits.None, t_profile, _new_phase_control[dof], MaxVelocity[dof], _inp_min_velocity[dof], MaxAcceleration[dof], _inp_min_acceleration[dof], MaxJerk[dof])
                THEN
                  found_time_synchronization := FALSE;                        
                END_IF
              ELSIF NOT IsInfinity(MaxAcceleration[dof])
              THEN
                IF NOT p.CheckForSecondOrderWithTiming2(ProfileControlSigns.Uddu, ReachedLimits.None, t_profile, _new_phase_control[dof], -_new_phase_control[dof], MaxVelocity[dof], _inp_min_velocity[dof], MaxAcceleration[dof], _inp_min_acceleration[dof])
                THEN
                  found_time_synchronization := FALSE;                        
                END_IF
              ELSE
                IF NOT p.CheckForFirstOrderWithTiming2(ProfileControlSigns.Uddu, ReachedLimits.None, t_profile, _new_phase_control[dof], MaxVelocity[dof], _inp_min_velocity[dof])
                THEN
                  found_time_synchronization := FALSE;                        
                END_IF
              END_IF
            
            ProfileControlSigns.Udud:
              IF NOT IsInfinity(MaxJerk[dof])
              THEN            
                IF NOT p.CheckWithTiming2(ProfileControlSigns.Udud, ReachedLimits.None, t_profile, _new_phase_control[dof], MaxVelocity[dof], _inp_min_velocity[dof], MaxAcceleration[dof], _inp_min_acceleration[dof], MaxJerk[dof])
                THEN            
                  found_time_synchronization := FALSE;
                END_IF
              ELSE
                IF NOT p.CheckForSecondOrderWithTiming2(ProfileControlSigns.Udud, ReachedLimits.None, t_profile, _new_phase_control[dof], -_new_phase_control[dof], MaxVelocity[dof], _inp_min_velocity[dof], MaxAcceleration[dof], _inp_min_acceleration[dof])
                THEN
                  found_time_synchronization := FALSE;                        
                END_IF
              END_IF                
          END_CASE
        
        ControlInterfaceType.Velocity:
          CASE p.ControlSigns
          OF
            ProfileControlSigns.Uddu:
            
              IF NOT IsInfinity(MaxJerk[dof])
              THEN  
                IF NOT p.CheckForVelocityWithTiming(ProfileControlSigns.Uddu, ReachedLimits.None, _new_phase_control[dof], MaxAcceleration[dof], _inp_min_acceleration[dof], MaxJerk[dof])
                THEN
                  found_time_synchronization := FALSE;                        
                END_IF
              ELSE
                IF NOT p.CheckForSecondOrderVelocityWithTiming2(ProfileControlSigns.Uddu, ReachedLimits.None, t_profile, _new_phase_control[dof], MaxAcceleration[dof], _inp_min_acceleration[dof])
                THEN
                  found_time_synchronization := FALSE;                        
                END_IF
              END_IF
          
            ProfileControlSigns.Udud:
            
              IF NOT IsInfinity(MaxJerk[dof])
              THEN             
                IF NOT p.CheckForVelocityWithTiming(ProfileControlSigns.Udud, ReachedLimits.None, _new_phase_control[dof], MaxAcceleration[dof], _inp_min_acceleration[dof], MaxJerk[dof])
                THEN            
                  found_time_synchronization := FALSE;
                END_IF
              ELSE
                IF NOT p.CheckForSecondOrderVelocityWithTiming2(ProfileControlSigns.Udud, ReachedLimits.None, t_profile, _new_phase_control[dof], MaxAcceleration[dof], _inp_min_acceleration[dof])
                THEN
                  found_time_synchronization := FALSE;                        
                END_IF
              END_IF                
          END_CASE        
      END_CASE
  

      p.Limits := p_limiting.Limits; // After check method call to set correct limits
    END_FOR

    IF found_time_synchronization AND_THEN phaseOrNoneSychronizationCount = _dofsEnd  THEN
      RETURN;
    END_IF
  END_IF
END_IF

// Time Synchronization
FOR dof:=0 TO _dofsEnd
DO
  IF NOT Enabled[dof] OR_ELSE ((dof = limiting_dof OR_ELSE _inp_per_dof_synchronization[dof] = SynchronizationType.None) AND_THEN NOT discrete_duration) THEN
    CONTINUE;
  END_IF
  
  p REF= _profiles[dof];
  t_profile := Duration - p.Brake.Duration - p.Accel.Duration;
  
  IF (_inp_per_dof_synchronization[dof] = SynchronizationType.TimeIfNecessarySync AND_THEN ABS(TargetVelocity[dof]) < Constants.Epsilon AND_THEN ABS(CurrentAcceleration[dof]) < Constants.Epsilon) THEN
      p := _blocks[dof].Pmin;
      CONTINUE;
  END_IF
  
  // Check if the final time corresponds to an extremal profile calculated in step 1
  // Use 2*eps because of numerical robustness in duration discretization
  IF (ABS(t_profile - _blocks[dof].Tmin) < Constants.Epsilon) THEN
      p := _blocks[dof].Pmin;
      CONTINUE;
  ELSIF (_blocks[dof].A.IsUsed AND_THEN ABS(t_profile - _blocks[dof].A.Right) < 2 * Constants.Epsilon16)
  THEN
      p := _blocks[dof].A.Profile;
      CONTINUE;
  ELSIF (_blocks[dof].B.IsUsed AND_THEN ABS(t_profile - _blocks[dof].B.Right) < 2 * Constants.Epsilon16)
  THEN
      p := _blocks[dof].B.Profile;
      CONTINUE;
  END_IF
  
  CASE (_inp_per_dof_control_interface[dof])
  OF  
    ControlInterfaceType.Position: 
    
      IF NOT IsInfinity(MaxJerk[dof])
      THEN       
        _positionThirdOrderStep2.Set(t_profile, p.p[0], p.v[0], p.a[0], p.pf, p.vf, p.af, MaxVelocity[dof], _inp_min_velocity[dof], MaxAcceleration[dof], _inp_min_acceleration[dof], MaxJerk[dof]);
        found_time_synchronization := _positionThirdOrderStep2.Get(p);
      ELSIF NOT IsInfinity(MaxAcceleration[dof])
      THEN
        _positionSecondOrderStep2.Set(t_profile, p.p[0], p.v[0], p.pf, p.vf, MaxVelocity[dof], _inp_min_velocity[dof], MaxAcceleration[dof], _inp_min_acceleration[dof]);
        found_time_synchronization := _positionSecondOrderStep2.Get(p);        
      ELSE
        _positionFirstOrderStep2.Set(t_profile, p.p[0], p.pf, MaxVelocity[dof], _inp_min_velocity[dof]);
        found_time_synchronization := _positionFirstOrderStep2.Get(p);        
      END_IF

    ControlInterfaceType.Velocity: 
      IF NOT IsInfinity(MaxJerk[dof])
      THEN    
        _velocityThirdOrderStep2.Set(t_profile, p.v[0], p.a[0], p.vf, p.af, MaxAcceleration[dof], _inp_min_acceleration[dof], MaxJerk[dof]);
        found_time_synchronization := _velocityThirdOrderStep2.Get(p);
      ELSE
        _velocitySecondOrderStep2.Set(t_profile, p.v[0], p.vf, MaxAcceleration[dof], _inp_min_acceleration[dof]);
        found_time_synchronization := _velocitySecondOrderStep2.Get(p);
      END_IF
  END_CASE

  IF NOT found_time_synchronization
  THEN
    AbortErrorId(TrajectoryErrorCode.SynchronizationFailed, '');
    RETURN;
  END_IF
END_FOR
END_METHOD

/// This method simply calls the body of the function block
METHOD Cyclic
VAR_INPUT
END_VAR
THIS^();
END_METHOD

/// Total planned trajectory duration in seconds.
/// The value is set after successful calculation and remains valid until inputs
/// change or [Reset](xref:Struckig.Otg#Reset) is called.
///
/// In synchronized operation this is the common duration for all participating DoFs.
PROPERTY Duration : LREAL
GET
Duration := _duration;
END_GET
END_PROPERTY

/// Returns the current error code.
/// Use together with [ErrorMessage](xref:Struckig.Otg#ErrorMessage) for diagnostics.
METHOD ErrorCode : TrajectoryErrorCode
VAR_INPUT
END_VAR
ErrorCode := _errorId;
END_METHOD

/// Returns a human-readable error description.
/// If no custom error text exists, a default description is derived from
/// [ErrorCode](xref:Struckig.Otg#ErrorCode).
METHOD ErrorMessage : STRING(255)
VAR_INPUT
END_VAR
IF _errorMessage = ''
THEN
  CASE _errorId
  OF
    TrajectoryErrorCode.CalculateStep1Failed: ErrorMessage := 'Trajectory generation failed in step1';
    TrajectoryErrorCode.InvalidInput: ErrorMessage := 'Trajectory-generation invalid input';
    TrajectoryErrorCode.SynchronizationFailed: ErrorMessage := 'Trajectory-generation synchronization failed';
    TrajectoryErrorCode.ZeroLimitsConflict: ErrorMessage := 'Zero limits conflict in step 1';
    TrajectoryErrorCode.ZeroLimitsConflictInSynchronization: ErrorMessage := 'Zero limits conflict with other degrees of freedom in time synchronization';

  ELSE
    IF State = TrajectoryState.Error
    THEN
      ErrorMessage := 'Unknown error';
    END_IF
  END_CASE
ELSE
  ErrorMessage := _errorMessage;
END_IF
END_METHOD

METHOD FB_init : BOOL
VAR_INPUT
	bInitRetains : BOOL; // if TRUE, the retain variables are initialized (warm start / cold start)
	bInCopyCode : BOOL;  // if TRUE, the instance afterwards gets moved into the copy code (online change)
  cycletime : LREAL;
  dofs : SINT;
END_VAR
VAR
  i : INT;
  blockSize : UDINT := SIZEOF(Block)*SINT_TO_UDINT(dofs);
  profileSize : UDINT :=  SIZEOF(ProfileDesc)*SINT_TO_UDINT(dofs);  
END_VAR
THIS^.Dofs := dofs;

FOR i:=0 TO ParameterList.MaxDoFs
DO
  Enabled[i] := i < dofs;
  MaxAcceleration[i] := Constants.Infinity;  
  MaxJerk[i] := Constants.Infinity;
END_FOR
_dt := THIS^.CycleTime := cycletime;
END_METHOD

METHOD PRIVATE HasChanged : BOOL
VAR
  i : INT;  
END_VAR
IF _dofs <> Dofs
THEN
  HasChanged := TRUE;
  RETURN;
END_IF

FOR i:=0 TO _dofsEnd
DO
  IF NOT (_currentPosition[i] = CurrentPosition[i] AND_THEN
     _currentVelocity[i] = CurrentVelocity[i] AND_THEN
     _currentAcceleration[i] = CurrentAcceleration[i] AND_THEN
     _targetPosition[i] = TargetPosition[i] AND_THEN
     _targetVelocity[i] = TargetVelocity[i] AND_THEN
     _targetAcceleration[i] = TargetAcceleration[i] AND_THEN
     _maxVelocity[i] = MaxVelocity[i] AND_THEN
     _maxAcceleration[i] = MaxAcceleration[i] AND_THEN
     _maxJerk[i] = MaxJerk[i] AND_THEN
     _enabled[i] = Enabled[i] AND_THEN
     _minVelocity[i] = MinVelocity[i] AND_THEN
     _minAcceleration[i] = MinAcceleration[i] AND_THEN
     _perDofControlInterface[i] = PerDofControlInterface[i] AND_THEN
     _perDofSynchronization[i] = PerDofSynchronization[i])
  THEN
    HasChanged := TRUE;  
    RETURN;
	END_IF
END_FOR

IF NOT (_controlInterface = ControlInterface AND_THEN
   _synchronization = Synchronization AND_THEN
   _discretization = Discretization AND_THEN
   _minDuration = MinDuration AND_THEN
   _smoothBrake = SmoothBrake)   
THEN
  HasChanged := TRUE;
  RETURN;
END_IF
END_METHOD

METHOD INTERNAL IsBlocked : BOOL
VAR_INPUT
  block : REFERENCE TO Block;
  t : LREAL;
END_VAR
IsBlocked := (t < block.Tmin) OR_ELSE (block.A.IsUsed AND_THEN block.A.Left < t AND_THEN t < block.A.Right) OR_ELSE (block.B.IsUsed AND_THEN block.B.Left < t AND_THEN t < block.B.Right);
END_METHOD

/// Is the trajectory (in principle) phase synchronizable?
METHOD INTERNAL IsInputCollinear : BOOL
VAR_INPUT
  limitingDirection : ProfileDirection;
  limitingDof : INT;
  new_phase_control : REFERENCE TO ARRAY[0..ParameterList.MaxDoFs] OF LREAL;
END_VAR
VAR_INST
  scale_dof : INT := -1;
  dof : INT;
  pd : ARRAY[0..ParameterList.MaxDoFs] OF LREAL;
  scale_vector : POINTER TO LREAL;
  pd_scale, v0_scale, a0_scale, vf_scale, af_scale, scale, scale_limiting, current_scale : LREAL;
  control_limiting : LREAL;
END_VAR
// Check that vectors pd, v0, a0, vf, af are collinear
FOR dof:=0 TO _dofsEnd
DO
  pd[dof] := TargetPosition[dof] - CurrentPosition[dof];
END_FOR

scale_dof := -1;
FOR dof:=0 TO _dofsEnd
DO
  IF _inp_per_dof_synchronization[dof] <> SynchronizationType.Phase
  THEN
    CONTINUE;
	END_IF
  
  IF _inp_per_dof_control_interface[dof] = ControlInterfaceType.Position AND_THEN ABS(pd[dof]) > Constants.Epsilon
  THEN
    scale_vector := ADR(pd);
    scale_dof := dof;
    EXIT;

  ELSIF ABS(CurrentVelocity[dof]) > Constants.Epsilon
  THEN
    scale_vector := ADR(CurrentVelocity);
    scale_dof := dof;
    EXIT;

  ELSIF ABS(CurrentAcceleration[dof]) >  Constants.Epsilon
  THEN
    scale_vector := ADR(CurrentAcceleration);
    scale_dof := dof;
    EXIT;
  
  ELSIF ABS(TargetVelocity[dof]) >  Constants.Epsilon
  THEN
    scale_vector := ADR(TargetVelocity);
    scale_dof := dof;
    EXIT;

  ELSIF ABS(TargetAcceleration[dof]) > Constants.Epsilon
  THEN
    scale_vector := ADR(TargetAcceleration);
    scale_dof := dof;
    EXIT;
  END_IF
END_FOR

IF scale_dof < 0
THEN
  RETURN; // Zero everywhere is in theory collinear, but that trivial case is better handled elsewhere
END_IF

scale := scale_vector[scale_dof];
pd_scale := pd[scale_dof] / scale;
v0_scale := CurrentVelocity[scale_dof] / scale;
vf_scale := TargetVelocity[scale_dof] / scale;
a0_scale := CurrentAcceleration[scale_dof] / scale;
af_scale := TargetAcceleration[scale_dof] / scale;

scale_limiting := scale_vector[limitingDof];
control_limiting := SEL(limitingDirection = ProfileDirection.Up, -MaxJerk[limitingDof], MaxJerk[limitingDof]);

IF IsInfinity(MaxJerk[limitingDof])
THEN
  control_limiting := SEL(limitingDirection = ProfileDirection.Up, _inp_min_acceleration[limitingDof], MaxAcceleration[limitingDof]);
END_IF

IF ABS(scale_limiting) < Constants.Epsilon
THEN
  RETURN;
END_IF

FOR dof:=0 TO _dofsEnd
DO
  IF _inp_per_dof_synchronization[dof] <> SynchronizationType.Phase
  THEN
    CONTINUE;
	END_IF
  
  current_scale := scale_vector[dof];
  IF (_inp_per_dof_control_interface[dof] = ControlInterfaceType.Position AND_THEN ABS(pd[dof] - pd_scale * current_scale) > Constants.Epsilon)
    OR_ELSE ABS(CurrentVelocity[dof] - v0_scale * current_scale) > Constants.Epsilon
    OR_ELSE ABS(CurrentAcceleration[dof] - a0_scale * current_scale) > Constants.Epsilon
    OR_ELSE ABS(TargetVelocity[dof] - vf_scale * current_scale) > Constants.Epsilon
    OR_ELSE ABS(TargetAcceleration[dof] - af_scale * current_scale) > Constants.Epsilon
  THEN
    RETURN;
	END_IF
  
  new_phase_control[dof] := control_limiting * current_scale / scale_limiting;
END_FOR

IsInputCollinear := TRUE;
END_METHOD

/// Copies `NewPosition`, `NewVelocity`, and `NewAcceleration`
/// to the corresponding current-state inputs.
/// This helper connects one cycle output to the next cycle input and is useful
/// in closed-loop PLC applications.
///
/// Equivalent to manually assigning:
/// ```st
/// CurrentPosition := NewPosition;
/// CurrentVelocity := NewVelocity;
/// CurrentAcceleration := NewAcceleration;
/// ```
METHOD PassOutputToInput
VAR_INPUT
END_VAR
CurrentPosition := NewPosition;
CurrentVelocity := NewVelocity;
CurrentAcceleration := NewAcceleration;

// Remove first intermediate waypoint if section did change
// not supported in Struckig, this is a Ruckig Pro Feature
//IF HasSectionChanged AND_THEN IntermediatePositionCount > 0
//THEN
//  IntermediatePositionIndex := IntermediatePositionIndex + 1;
//END_IF
END_METHOD

/// Resets the instance (e.g. to force a new calculation on the next update).
/// This method can be used to trigger a new trajectory even if inputs do not change.
/// Use this when external state jumps occur (manual jog, homing, drive reset)
/// and the generator must reinitialize from the new measured state.
METHOD Reset
VAR_INPUT
END_VAR
_inputInitialized := FALSE;
END_METHOD

METHOD PROTECTED SetBusy
VAR_INPUT
  on : BOOL;
END_VAR
_state := TrajectoryState.Busy;
END_METHOD

/// Current state of the trajectory generator.
/// - `Busy`: active trajectory is running.
/// - `Idle`: trajectory reached end state.
/// - `Error`: invalid input or unsynchronizable profile.
///
/// Check this property to decide whether to continue commanding setpoints,
/// hold final values, or handle a fault.
PROPERTY State : TrajectoryState
GET
State := _state;
END_GET
END_PROPERTY

METHOD INTERNAL Synchronize : BOOL
VAR_INPUT
  discrete_duration : BOOL;
END_VAR
VAR_IN_OUT
  Tmin : LREAL;
  t_sync : LREAL;
  limiting_dof : INT;
END_VAR
VAR_INST
  possible_t_syncs : ARRAY [0..3*ParameterList.MaxDoFs] OF LREAL;
  idx : ARRAY [0..3*ParameterList.MaxDoFs] OF INT;  
  idx_end : INT;
  possible_t_sync : REFERENCE TO LREAL;
  any_interval : BOOL;
  dof : INT;
  i,j, h : INT;
  is_blocked : BOOL;
  remainder : LREAL;
END_VAR
// Possible t_syncs are the start times of the intervals and optional Tmin
any_interval := FALSE;
FOR dof := 0 TO _dofsEnd
DO
  // Ignore DoFs without synchronization here
  IF _inp_per_dof_synchronization[dof] = SynchronizationType.None
  THEN
    possible_t_syncs[dof] := 0;
    possible_t_syncs[Dofs + dof] := Constants.Infinity;
    possible_t_syncs[2 * Dofs + dof] := Constants.Infinity;
  ELSE
    possible_t_syncs[dof] := _blocks[dof].Tmin;
    possible_t_syncs[Dofs + dof] := SEL(_blocks[dof].A.IsUsed, Constants.Infinity, _blocks[dof].A.Right);
    possible_t_syncs[2 * Dofs + dof] := SEL(_blocks[dof].B.IsUsed, Constants.Infinity, _blocks[dof].B.Right);
    any_interval := any_interval OR_ELSE _blocks[dof].A.IsUsed OR_ELSE _blocks[dof].B.IsUsed;
  END_IF
END_FOR

possible_t_syncs[3 * Dofs] := SEL(Tmin = 0, Tmin, Constants.Infinity);
any_interval := any_interval OR_ELSE Tmin > 0;
IF discrete_duration
THEN
  FOR i:=0 TO 3*Dofs-1
  DO
    possible_t_sync REF= possible_t_syncs[i];
    IF possible_t_sync = Constants.Infinity
    THEN
      CONTINUE;
		END_IF
    
    remainder := Fmod(possible_t_sync, CycleTime); // in [0, delta_time)
    IF remainder > Constants.Epsilon16 THEN
      possible_t_sync := possible_t_sync + CycleTime - remainder;
    END_IF     
  END_FOR
END_IF

// Bubblesort possible_t_syncs from best to worst
idx_end := SEL(any_interval, _dofsEnd, 3*DOFs);
BubbleSortLreal(ADR(possible_t_syncs), idx_end, indicesSorted:=ADR(idx));

// Start at last tmin (or worse)
FOR i:=_dofsEnd TO idx_end
DO  
  possible_t_sync REF= possible_t_syncs[idx[i]];
  
  is_blocked := FALSE;
  FOR dof:=0 TO _dofsEnd
  DO
    IF _inp_per_dof_synchronization[dof] = SynchronizationType.None
    THEN
      CONTINUE;
		END_IF
    
    IF IsBlocked(_blocks[dof], possible_t_sync) 
    THEN
      is_blocked := TRUE;
      EXIT;
		END_IF
	END_FOR
  
  IF is_blocked OR_ELSE possible_t_sync < Tmin OR_ELSE possible_t_sync = Constants.Infinity
  THEN
    CONTINUE;
	END_IF
    
  t_sync := possible_t_sync;
  IF (idx[i] = 3*Dofs)  // Optional Tmin
  THEN
    limiting_dof := -1;
    Synchronize := TRUE;
    RETURN;
  END_IF

  limiting_dof := (idx[i] MOD Dofs);
  CASE TRUNC(idx[i] / Dofs)
  OF
    0: _profiles[limiting_dof] := _blocks[limiting_dof].Pmin;
    1: _profiles[limiting_dof] := _blocks[limiting_dof].A.Profile;
    2: _profiles[limiting_dof] := _blocks[limiting_dof].B.Profile;  
	END_CASE
  
  Synchronize := TRUE;
  RETURN;
  
END_FOR
END_METHOD

/// To check that *Struckig* is able to generate a trajectory before the actual calculation step,
/// ```st
/// ruckig.ValidateInput(input, currentState: FALSE, targetState: TRUE);
/// // returns boolean
/// ```
/// returns `FALSE` if an input is not valid. The two boolean arguments check that the current or target state are 
/// within the limits. The check includes a typical catch of jerk-limited trajectory generation: 
/// When the current state is at maximal velocity, any positive acceleration will inevitable lead to a velocity violation 
/// *at a future timestep*. In general, this condition is fulfilled when
/// ```
/// Abs(acceleration) <= Sqrt(2 * max_jerk * (max_velocity - Abs(velocity))).
/// ```
/// If both arguments are set to true, the calculated trajectory is guaranteed to be *within the kinematic limits throughout* 
/// its duration. Also, note that there are range constraints of the input due to numerical reasons, see below for more details.
///
/// Recommended usage before applying new targets:
/// ```st
/// IF otg.ValidateInput(TRUE, TRUE) THEN
///   // inputs are valid, call cyclic calculation
///   otg();
/// ELSE
///   // inspect otg.ErrorCode() and otg.ErrorMessage()
/// END_IF
/// ```
{attribute 'conditionalshow'}
METHOD ValidateInput : BOOL
VAR_INPUT
  checkCurrentStateWithinLimits : BOOL;
  checkTargetStateWithinLimits : BOOL;
END_VAR
VAR
  stateMem : TrajectoryState;
END_VAR
stateMem := _state;
ValidateInput := ValidateInputOrAbort(checkCurrentStateWithinLimits, checkTargetStateWithinLimits);
_state := stateMem;
END_METHOD

/// \copydoc Struckig.Otg#ValidateInput
{attribute 'conditionalshow'}
METHOD PROTECTED ValidateInputOrAbort : BOOL
VAR_INPUT
  checkCurrentStateWithinLimits : BOOL;
  checkTargetStateWithinLimits : BOOL;
END_VAR
VAR
  i, dofsEnd : INT;
  aMin, vMin, a0, af, v0, vf : LREAL;
  ci : ControlInterfaceType;
END_VAR
IF Dofs = 0
THEN
  RETURN;
END_IF

dofsEnd := Dofs-1;
FOR i:=0 TO dofsEnd
DO

  IF MaxJerk[i] <> MaxJerk[i] OR_ELSE // isnan
     MaxJerk[i] < 0.0
  THEN
    AbortErrorId(TrajectoryErrorCode.InvalidInput, 'maximum jerk limit should be larger than or equal to zero');
    RETURN;
	END_IF

  IF MaxAcceleration[i] <> MaxAcceleration[i] OR_ELSE // isnan
     MaxAcceleration[i] < 0.0
  THEN
    AbortErrorId(TrajectoryErrorCode.InvalidInput, 'maximum acceleration limit should be larger than or equal to zero'); 
    RETURN;
  END_IF

  aMin := SEL(MinAcceleration[i] = 0, MinAcceleration[i] ,-MaxAcceleration[i]);
  IF aMin <> aMin OR_ELSE // isnan  
     aMin > 0
  THEN    
    AbortErrorId(TrajectoryErrorCode.InvalidInput, 'minimum acceleration limit should be smaller than or equal zero'); 
    RETURN;
  END_IF
  
  a0 := CurrentAcceleration[i];
  IF a0 <> a0 // isnan
  THEN
    AbortErrorId(TrajectoryErrorCode.InvalidInput, 'current acceleration should be a valid number'); 
    RETURN;
	END_IF
  
  af := TargetAcceleration[i];
  IF af <> af // isnan
  THEN
    AbortErrorId(TrajectoryErrorCode.InvalidInput, 'target acceleration should be a valid number'); 
    RETURN;
	END_IF  
  
  IF checkCurrentStateWithinLimits
  THEN
    IF a0 > MaxAcceleration[i]
    THEN
      AbortErrorId(TrajectoryErrorCode.InvalidInput, 'current acceleration exceeds its maximum acceleration limit'); 
      RETURN;
    END_IF
    
    IF  a0 < aMin
    THEN 
      AbortErrorId(TrajectoryErrorCode.InvalidInput, 'current acceleration undercuts its minimum acceleration limit'); 
      RETURN;
    END_IF    
  END_IF
  
  IF checkTargetStateWithinLimits 
  THEN
    IF af > MaxAcceleration[i]
    THEN
      AbortErrorId(TrajectoryErrorCode.InvalidInput, 'target acceleration exceeds its maximum acceleration limit'); 
      RETURN;
    END_IF
 
    IF af < aMin
    THEN
      AbortErrorId(TrajectoryErrorCode.InvalidInput, 'target acceleration undercuts its minimum acceleration limit'); 
      RETURN;  
		END_IF
  END_IF
  
  v0 := CurrentVelocity[i];
  IF v0 <> v0// isnan
  THEN
    AbortErrorId(TrajectoryErrorCode.InvalidInput, 'current velocity should be a valid number'); 
    RETURN;
	END_IF
  
  vf := TargetVelocity[i];
  IF vf <> vf // isnan
  THEN
    AbortErrorId(TrajectoryErrorCode.InvalidInput, 'target velocity should be a valid number'); 
    RETURN;
	END_IF
  
  ci := SEL(PerDofControlInterface[i] = ControlInterfaceType.Undefined, PerDofControlInterface[i], ControlInterface);
  IF (ci = ControlInterfaceType.Position)
  THEN
  
    IF CurrentPosition[i] <> CurrentPosition[i] //isnan
    THEN
      AbortErrorId(TrajectoryErrorCode.InvalidInput, 'current position should be a valid number'); 
      RETURN;
    END_IF
    
    IF TargetPosition[i] <> TargetPosition[i] //isnan
    THEN
      AbortErrorId(TrajectoryErrorCode.InvalidInput, 'target position should be a valid number'); 
      RETURN;
    END_IF    
    
    IF MaxVelocity[i] <> MaxVelocity[i] OR_ELSE // isnan
       MaxVelocity[i] < 0.0      
    THEN
      AbortErrorId(TrajectoryErrorCode.InvalidInput, 'maximum velocity limit should be larger than or equal to zero'); 
      RETURN;
		END_IF
    
    vMin := SEL(MinVelocity[i] = 0, MinVelocity[i], -MaxVelocity[i]);
    IF vMin <> vMin OR_ELSE // isnan
       vMin > 0.0
    THEN
      AbortErrorId(TrajectoryErrorCode.InvalidInput, 'minimum velocity limit should be smaller than or equal to zero'); 
      RETURN;
    END_IF
    
    IF checkCurrentStateWithinLimits 
    THEN
      IF v0 > MaxVelocity[i]
      THEN
        AbortErrorId(TrajectoryErrorCode.InvalidInput, 'current velocity exceeds its maximum velocity limit'); 
        RETURN;
      END_IF

      IF v0 < vMin
      THEN
        AbortErrorId(TrajectoryErrorCode.InvalidInput, 'current velocity undercuts its minimum velocity limit'); 
        RETURN;
      END_IF
    END_IF
    
    IF checkTargetStateWithinLimits
    THEN
      IF vf > MaxVelocity[i]
      THEN
        AbortErrorId(TrajectoryErrorCode.InvalidInput, 'target velocity exceeds its maximum velocity limit'); 
        RETURN;
      END_IF
      
      IF vf < vMin
      THEN
        AbortErrorId(TrajectoryErrorCode.InvalidInput, 'target velocity undercuts its minimum velocity limit'); 
        RETURN;
			END_IF
    END_IF
    
    IF checkCurrentStateWithinLimits
    THEN
      IF a0 > 0 AND_THEN MaxJerk[i] > 0 AND_THEN VelocityAtZero(v0, a0, MaxJerk[i]) > MaxVelocity[i]
      THEN
        AbortErrorId(TrajectoryErrorCode.InvalidInput, 'Trajectory will inevitably reach a velocity from the current kinematic state that will exceed its maximum velocity limit'); 
        RETURN;
			END_IF
      
      IF a0 < 0 AND_THEN MaxJerk[i] > 0 AND_THEN VelocityAtZero(v0, a0, -MaxJerk[i]) < vMin
      THEN
        AbortErrorId(TrajectoryErrorCode.InvalidInput, 'Trajectory will inevitably reach a velocity from the current kinematic state that will undercut its minimum velocity limit'); 
        RETURN;
			END_IF      
    END_IF
    
    IF checkTargetStateWithinLimits
    THEN
      IF af < 0 AND_THEN MaxJerk[i] > 0 AND_THEN VelocityAtZero(vf, af, MaxJerk[i]) > MaxVelocity[i]
      THEN
        AbortErrorId(TrajectoryErrorCode.InvalidInput, 'Trajectory will inevitably reach a velocity from the current kinematic state that will exceed its maximum velocity limit'); 
        RETURN;
			END_IF
      
      IF af > 0 AND_THEN MaxJerk[i] > 0 AND_THEN VelocityAtZero(vf, af, -MaxJerk[i]) < vMin
      THEN
        AbortErrorId(TrajectoryErrorCode.InvalidInput, 'Trajectory will inevitably reach a velocity from the current kinematic state that will undercut its minimum velocity limit'); 
        RETURN;
			END_IF  
    END_IF    
  END_IF

END_FOR

IF CycleTime <= 0 AND_THEN Discretization <> DiscretizationType.Continuous
THEN
  AbortErrorId(TrajectoryErrorCode.InvalidInput, 'Cycle time parameter should be larger than zero'); 
  RETURN;
END_IF

ValidateInputOrAbort := TRUE;
END_METHOD

METHOD INTERNAL VelocityAtZero : LREAL
VAR_INPUT
  v0 : LREAL;
  a0 : LREAL;
  j : LREAL;
END_VAR
VelocityAtZero := v0 + (a0 * a0)/(2 * j);
END_METHOD

END_FUNCTION_BLOCK

// ---- Struckig/Profile/ProfileDesc.TcPOU
// Struckig
// Copyright (C) 2022 Stefan Besler

// This program is free software: you can redistribute it and/or modify
// it under the terms of the GNU General Public License as published by
// the Free Software Foundation, either version 3 of the License, or
// (at your option) any later version.

// This program is distributed in the hope that it will be useful,
// but WITHOUT ANY WARRANTY; without even the implied warranty of
// MERCHANTABILITY or FITNESS FOR A PARTICULAR PURPOSE.  See the
// GNU General Public License for more details.
//
// You should have received a copy of the GNU General Public License
// along with THIS PROGRAM.  IF NOT, see <http://www.gnu.org/licenses/>.
/// The state Profile for position, velocity, acceleration and jerk for a single DoF
/// A single-dof kinematic profile with position, velocity, acceleration and jerk
{attribute 'hide'}
FUNCTION_BLOCK ProfileDesc
VAR_INPUT
  Limits : ReachedLimits;
  Direction : ProfileDirection;
  ControlSigns : ProfileControlSigns;
  
  t, t_sum, j : ARRAY[0..6] OF LREAL;
  a, v, p : ARRAY[0..7] OF LREAL;

  pf, vf, af : LREAL; //! Target (final) kinematic state
  Brake, Accel : BrakeProfile; //! Brake sub-profiles
END_VAR

METHOD Bound : ProfileBound
VAR_INPUT
END_VAR
VAR
  i : INT;
  t_current_sum : LREAL;
END_VAR
Bound.Minimum := Constants.Infinity;
Bound.Maximum := -Constants.Infinity;

IF Brake.Duration > 0.0
THEN
  IF (Brake.t[0] > 0.0)
  THEN
    CheckStepForBound(0.0, Brake.t[0], Brake.p[0], Brake.v[0], Brake.a[0], Brake.j[0], Bound);
  
    IF (Brake.t[1] > 0.0) 
    THEN
      CheckStepForBound(Brake.t[0], Brake.t[1], Brake.p[1], Brake.v[1], Brake.a[1], Brake.j[1], Bound);
      
      IF (Brake.t[2] > 0.0)
      THEN
        CheckStepForBound(Brake.t[0] + Brake.t[1], Brake.t[2], Brake.p[2], Brake.v[2], Brake.a[2], Brake.j[2], Bound);
      END_IF
    END_IF
  END_IF
END_IF

t_current_sum := 0;        
FOR i:=0 TO 6
DO
  IF i > 0
  THEN
    t_current_sum := t_sum[i-1];
	END_IF
  
  CheckStepForBound(t_current_sum + Brake.Duration, t[i], p[i], v[i], a[i], j[i], Bound);
END_FOR 

IF (pf < Bound.Minimum)
THEN
  Bound.Minimum := pf;
  Bound.Tmin := t_sum[6] + Brake.Duration;
END_IF 


IF (pf > Bound.Maximum) 
THEN
  Bound.Maximum := pf;
  Bound.Tmax := t_sum[6] + Brake.Duration;
END_IF
END_METHOD

METHOD CheckBound : BOOL
VAR_INPUT
  t_ext, t_sum, t, p, v, a, j : LREAL;
END_VAR
VAR_IN_OUT
  b : ProfileBound;     
END_VAR
VAR
  p_ext, v_Ext, a_ext : LREAL;
END_VAR
IF (0 < t_ext AND_THEN t_ext < t)
THEN
  Integrate(t_ext, p, v, a, j, p:=p_ext, v:=v_ext, a:=a_ext);
  IF (a_ext > 0 AND_THEN p_ext < b.Minimum)
  THEN
    b.Minimum := p_ext;
    b.Tmin := t_sum + t_ext;
   ELSIF (a_ext < 0 AND_THEN p_ext > b.Maximum) 
   THEN
    b.Maximum := p_ext;
    b.Tmax := t_sum + t_ext; 
  END_IF
END_IF
END_METHOD

/// For velocity interface
METHOD CheckForFirstOrder : BOOL
VAR_INPUT
  controlSigns : ProfileControlSigns;
  limits : ReachedLimits;  
  vUp : LREAL;
END_VAR
VAR
  i : INT;
  vUppLim : LREAL;
  vLowLim : LREAL;
  v_a_zero : LREAL;
END_VAR
// ReachedLimits::VEL
IF t[3] < 0.0
THEN
  RETURN;
END_IF

t_sum[0] := 0;
t_sum[1] := 0;
t_sum[2] := 0;
t_sum[3] := t[3];
t_sum[4] := t[3];
t_sum[5] := t[3];
t_sum[6] := t[3];

IF t_sum[6] > Constants.Tmax // For numerical reasons, is that needed?}
THEN
  RETURN;        
END_IF

j[0] := 0;
j[1] := 0;
j[2] := 0;
j[3] := 0;
j[4] := 0;
j[5] := 0;
j[6] := 0;

a[0] := 0;
a[1] := 0;
a[2] := 0;
a[3] := 0;
a[4] := 0;
a[5] := 0;
a[6] := 0;
a[7] := af;

v[0] := 0;
v[1] := 0;
v[2] := 0;
v[3] := SEL(t[3] > 0, 0, vUp);
v[4] := 0;
v[5] := 0;
v[6] := 0;
v[7] := vf;

FOR i:= 0 TO 6 
DO
  p[i+1] := p[i] + t[i] * (v[i] + t[i] * a[i] / 2);
END_FOR

THIS^.Direction := SEL(vUp > 0, ProfileDirection.Down, ProfileDirection.Up);
THIS^.ControlSigns := controlSigns;
THIS^.Limits := limits;

// Velocity limit can be broken in the beginning if both initial velocity and acceleration are too high
CheckForFirstOrder := ABS(p[7] - pf) < Constants.PositionPrecision;
END_METHOD

/// For velocity interface
METHOD CheckForFirstOrderWithTiming : BOOL
VAR_INPUT
  controlSigns : ProfileControlSigns;
  limits : ReachedLimits;  
  vUp : LREAL;
END_VAR
VAR
  i : INT;
  aUppLim : LREAL;
  aLowLim : LREAL;
END_VAR
CheckForFirstOrderWithTiming := CheckForFirstOrder(controlSigns, limits, vUp); // AND_THEN (ABS(t[6] - tf) < t_precision);
END_METHOD

/// For velocity interface
METHOD CheckForFirstOrderWithTiming2 : BOOL
VAR_INPUT
  controlSigns : ProfileControlSigns;
  limits : ReachedLimits;  
  tf : LREAL;
  vUp : LREAL;
  vMax, vMin : LREAL;
END_VAR
CheckForFirstOrderWithTiming2 :=
  (vMin - Constants.VelocityEpsilon < vUp)
  AND_THEN (vUp < vMax + Constants.VelocityEpsilon)
  AND_THEN CheckForFirstOrderWithTiming(controlSigns, limits, vUp);
END_METHOD

/// For velocity interface
METHOD CheckForSecondOrder : BOOL
VAR_INPUT
  controlSigns : ProfileControlSigns;
  limits : ReachedLimits;  
  aUp, aDown : LREAL;
  vMax, vMin : LREAL;
END_VAR
VAR
  i : INT;
  vUppLim : LREAL;
  vLowLim : LREAL;
  v_a_zero : LREAL;
END_VAR
// ReachedLimits::ACC0
IF t[0] < 0.0
THEN
  RETURN;
END_IF

t_sum[0] := t[0];
FOR i:=0 TO 5
DO
  IF (t[i+1] < 0)
  THEN
    RETURN;
  END_IF
  
  t_sum[i+1] := t_sum[i] + t[i+1];  
END_FOR

IF t_sum[6] > Constants.Tmax // For numerical reasons, is that needed?}
THEN
  RETURN;        
END_IF

j[0] := 0;
j[1] := 0;
j[2] := 0;
j[3] := 0;
j[4] := 0;
j[5] := 0;
j[6] := 0;

IF controlSigns = ProfileControlSigns.Uddu
THEN
  a[0] := SEL(t[0] > 0, 0, aUp);
  a[1] := 0;
  a[2] := SEL(t[2] > 0, 0, aDown);
  a[3] := 0;
  a[4] := SEL(t[4] > 0, 0, aDown);
  a[5] := 0;
  a[6] := SEL(t[6] > 0, 0, aUp);
  a[7] := af;
ELSE
  a[0] := SEL(t[0] > 0, 0, aUp);
  a[1] := 0;
  a[2] := SEL(t[2] > 0, 0, aDown);
  a[3] := 0;
  a[4] := SEL(t[4] > 0, 0, aUp);
  a[5] := 0;
  a[6] := SEL(t[6] > 0, 0, aDown);
  a[7] := af;
END_IF

direction := SEL(vMax > 0, ProfileDirection.Down, ProfileDirection.Up);
vUppLim := SEL(direction = ProfileDirection.Up, vMin, vMax) + Constants.VelocityEpsilon;
vLowLim := SEL(direction = ProfileDirection.Up, vMax, vMin) - Constants.VelocityEpsilon;

FOR i:= 0 TO 6 
DO
  v[i+1] := v[i] + t[i] * a[i];
  p[i+1] := p[i] + t[i] * (v[i] + t[i] * a[i] / 2);
END_FOR


THIS^.ControlSigns := controlSigns;
THIS^.Limits := limits;

// Velocity limit can be broken in the beginning if both initial velocity and acceleration are too high
CheckForSecondOrder := ABS(p[7] - pf) < Constants.PositionPrecision AND_THEN ABS(v[7] - vf) < Constants.VelocityPrecision
    AND_THEN v[2] <= vUppLim AND_THEN v[3] <= vUppLim AND_THEN v[4] <= vUppLim AND_THEN v[5] <= vUppLim AND_THEN v[6] <= vUppLim
    AND_THEN v[2] >= vLowLim AND_THEN v[3] >= vLowLim AND_THEN v[4] >= vLowLim AND_THEN v[5] >= vLowLim AND_THEN v[6] >= vLowLim;
END_METHOD

/// For velocity interface
METHOD CheckForSecondOrderVelocity : BOOL
VAR_INPUT
  controlSigns : ProfileControlSigns;
  limits : ReachedLimits;  
  aUp : LREAL;
END_VAR
VAR
  i : INT;
  aUppLim : LREAL;
  aLowLim : LREAL;
END_VAR
// ReachedLimits::ACC0
IF t[1] < 0.0
THEN
  RETURN;
END_IF

t_sum[0] := 0;
t_sum[1] := t[1];
t_sum[2] := t[1];
t_sum[3] := t[1];
t_sum[4] := t[1];
t_sum[5] := t[1];
t_sum[6] := t[1];

// For numerical reasons, is that needed?
IF t_sum[6] > Constants.Tmax
THEN
  RETURN;
END_IF


j[0] := 0;
j[1] := 0;
j[2] := 0;
j[3] := 0;
j[4] := 0;
j[5] := 0;
j[6] := 0;

a[0] := 0;
a[1] := aUp;
a[2] := 0;
a[3] := 0;
a[4] := 0;
a[5] := 0;
a[6] := 0;
a[7] := THIS^.af;

FOR i:=0 TO 6
DO
  v[i+1] := v[i] + t[i] * a[i];
  p[i+1] := p[i] + t[i] * (v[i] + t[i] * a[i] / 2);
END_FOR

THIS^.ControlSigns := controlSigns;
THIS^.Limits := limits;
THIS^.Direction := SEL(aUp > 0, ProfileDirection.Down, ProfileDirection.Up);

// Velocity limit can be broken in the beginning if both initial velocity and acceleration are too high
CheckForSecondOrderVelocity := ABS(v[6] - vf) < Constants.VelocityPrecision;
END_METHOD

/// For velocity interface
METHOD CheckForSecondOrderVelocityWithTiming : BOOL
VAR_INPUT
  controlSigns : ProfileControlSigns;
  limits : ReachedLimits;  
  aUp : LREAL;
END_VAR
CheckForSecondOrderVelocityWithTiming := CheckForSecondOrderVelocity(controlSigns, limits, aUp); // AND_THEN (ABS(t[6] - tf) < t_precision);
END_METHOD

/// For velocity interface
METHOD CheckForSecondOrderVelocityWithTiming2 : BOOL
VAR_INPUT
  controlSigns : ProfileControlSigns;
  limits : ReachedLimits;  
  tf : LREAL;
  aUp : LREAL;
  aMax : LREAL;
  aMin : LREAL;
END_VAR
CheckForSecondOrderVelocityWithTiming2 :=
 (aMin - Constants.AccelerationEpsilon < aUp)
 AND_THEN (aUp < aMax + Constants.AccelerationEpsilon)
 AND_THEN CheckForSecondOrderVelocityWithTiming(controlSigns, limits, aUp); // AND_THEN (ABS(t[6] - tf) < t_precision);
END_METHOD

/// For velocity interface
METHOD CheckForSecondOrderWithTiming : BOOL
VAR_INPUT
  controlSigns : ProfileControlSigns;
  limits : ReachedLimits;  
  tf : LREAL;
  aUp, aDown : LREAL;
  vMax, vMin : LREAL;
END_VAR
CheckForSecondOrderWithTiming := CheckForSecondOrder(controlSigns, limits, aUp, aDown, vMax, vMin);
END_METHOD

/// For velocity interface
METHOD CheckForSecondOrderWithTiming2 : BOOL
VAR_INPUT
  controlSigns : ProfileControlSigns;
  limits : ReachedLimits;  
  tf : LREAL;
  aUp, aDown : LREAL;
  vMax, vMin : LREAL;
  aMax, aMin : LREAL;  
END_VAR
CheckForSecondOrderWithTiming2 := 
    (aMin - Constants.AccelerationEpsilon < aUp)
    AND_THEN (aUp < aMax + Constants.AccelerationEpsilon)
    AND_THEN (aMin - Constants.AccelerationEpsilon < aDown)
    AND_THEN (aDown < aMax + Constants.AccelerationEpsilon)
    AND_THEN CheckForSecondOrderWithTiming(controlSigns, limits,tf, aUp, aDown, vMax, vMin);
END_METHOD

/// For velocity interface
METHOD CheckForVelocity : BOOL
VAR_INPUT
  controlSigns : ProfileControlSigns;
  limits : ReachedLimits;  
  jf : LREAL;
  aMax : LREAL;
  aMin : LREAL;  
END_VAR
VAR
  i : INT;
  aUppLim : LREAL;
  aLowLim : LREAL;
END_VAR
IF (t[0] < 0)
THEN
  RETURN;
END_IF

t_sum[0] := t[0];
FOR i:=0 TO 5
DO
  IF (t[i+1] < 0)
  THEN
    RETURN;
  END_IF
  
  t_sum[i+1] := t_sum[i] + t[i+1];
END_FOR


IF limits = ReachedLimits.Acc0
THEN
  IF t[1] < Constants.DoubleEpsilon
  THEN
    RETURN;
  END_IF
END_IF


IF t_sum[6] > Constants.Tmax // For numerical reasons, is that needed?}
THEN
  RETURN;        
END_IF

IF controlSigns = ProfileControlSigns.Uddu
THEN
  j[0] := SEL(t[0] > 0, 0, jf);
  j[1] := 0;
  j[2] := SEL(t[2] > 0, 0, -jf);
  j[3] := 0;
  j[4] := SEL(t[4] > 0, 0, -jf);
  j[5] := 0;
  j[6] := SEL(t[6] > 0, 0, jf);          
ELSE
  j[0] := SEL(t[0] > 0, 0, jf);
  j[1] := 0;
  j[2] := SEL(t[2] > 0, 0, -jf);
  j[3] := 0;
  j[4] := SEL(t[4] > 0, 0, jf);
  j[5] := 0;
  j[6] := SEL(t[6] > 0, 0, -jf); 
END_IF


FOR i:=0 TO 6
DO
  a[i+1] := a[i] + t[i] * j[i];
  v[i+1] := v[i] + t[i] * (a[i] + t[i] * j[i] / 2);
  p[i+1] := p[i] + t[i] * (v[i] + t[i] * (a[i] / 2 + t[i] * j[i] / 6));        
END_FOR

      
THIS^.ControlSigns := controlSigns;
THIS^.Limits := limits;

aUppLim := SEL((aMax > 0), aMin, aMax) + 5E-12;
aLowLim := SEL((aMax > 0), aMax, aMin) - 5E-12;

// Velocity limit can be broken in the beginning if both initial velocity and acceleration are too high
CheckForVelocity := ABS(v[7] - vf) < Constants.VelocityPrecision
    AND_THEN ABS(a[7] - af) < Constants.AccelerationPrecision // This is not really needed, but we want to double check
    AND_THEN a[1] >= aLowLim AND_THEN a[3] >= aLowLim AND_THEN a[5] >= aLowLim
    AND_THEN a[1] <= aUppLim AND_THEN a[3] <= aUppLim AND_THEN a[5] <= aUppLim;
END_METHOD

/// For velocity interface
METHOD CheckForVelocityWithTiming : BOOL
VAR_INPUT
  controlSigns : ProfileControlSigns;
  limits : ReachedLimits;  
  jf : LREAL;
  aMax : LREAL;
  aMin : LREAL;  
  jMax : LREAL;  
END_VAR
// Time doesn't need to be checked as every profile has a: tf - ... equation
CheckForVelocityWithTiming := (ABS(jf) < ABS(jMax) + Constants.JerkEpsilon) AND_THEN CheckForVelocity(controlSigns, limits, jf, aMax, aMin);
END_METHOD

METHOD CheckStepForBound : BOOL
VAR_INPUT
  t_sum, t, p, v, a, j : LREAL;
END_VAR
VAR_IN_OUT
  b : ProfileBound;  
END_VAR
VAR
  d, d_sqrt : LREAL;
END_VAR
IF (p < b.Minimum)
THEN 
  b.Minimum := p;
  b.Tmin := t_sum;
END_IF

IF (p > b.Maximum)
THEN 
  b.Maximum := p;
  b.Tmax := t_sum;
END_IF

IF (j <> 0) 
THEN
  d := a * a - 2 * j * v;
  IF (ABS(d) < Constants.DoubleEpsilon)
  THEN
    CheckBound(-a / j, t_sum, t, p, v, a, j, b:=b);
   ELSIF (d > 0) 
   THEN
    d_sqrt := SQRT(d);
    CheckBound((-a - D_sqrt) / j, t_sum, t, p, v, a, j, b:=b);
    CheckBound((-a + D_sqrt) / j, t_sum, t, p, v, a, j, b:=b);           
  END_IF
END_IF
END_METHOD

/// For position interface
METHOD CheckVel : BOOL
VAR_INPUT
  controlSigns : ProfileControlSigns;    
  limits : ReachedLimits;
  jf : LREAL;
  vMax : LREAL;
  vMin : LREAL;  
  aMax : LREAL;
  aMin : LREAL;
  setLimits : BOOL;
END_VAR
VAR
  i : INT;
  v_a_zero : LREAL;
  vUppLim, vLowLim : LREAL;  
  aUppLim, aLowLim : LREAL;
END_VAR
IF (t[0] < 0) 
THEN
  RETURN;
END_IF

t_sum[0] := t[0];
FOR i:=0 TO 5
DO
  IF (t[i+1] < 0)
  THEN
    RETURN;
  END_IF
  
  t_sum[i+1] := t_sum[i] + t[i+1];  
END_FOR

IF limits = ReachedLimits.Acc0Acc1Vel OR_ELSE limits = ReachedLimits.Acc0Vel OR_ELSE limits = ReachedLimits.Acc1Vel OR_ELSE limits = ReachedLimits.Vel THEN
  IF (t[3] < Constants.DoubleEpsilon) 
  THEN
    RETURN;                    
  END_IF
END_IF

IF limits = ReachedLimits.Acc0 OR_ELSE limits = ReachedLimits.Acc0Acc1
THEN
  IF (t[1] < Constants.DoubleEpsilon) 
  THEN
    RETURN;                    
  END_IF
END_IF

IF limits = ReachedLimits.Acc1 OR_ELSE limits = ReachedLimits.Acc0Acc1
THEN
  IF (t[5] < Constants.DoubleEpsilon)
  THEN
    RETURN;            
  END_IF
END_IF

IF t_sum[6] > Constants.Tmax  // For numerical reasons, is that needed?
THEN
  RETURN;        
END_IF
        
IF controlSigns = ProfileControlSigns.Uddu
THEN
  j[0] := SEL(t[0] > 0, 0, jf);
  j[1] := 0;
  j[2] := SEL(t[2] > 0, 0, -jf);
  j[3] := 0;
  j[4] := SEL(t[4] > 0, 0, -jf);
  j[5] := 0;
  j[6] := SEL(t[6] > 0, 0, jf);          
ELSE
  j[0] := SEL(t[0] > 0, 0, jf);
  j[1] := 0;
  j[2] := SEL(t[2] > 0, 0, -jf);
  j[3] := 0;
  j[4] := SEL(t[4] > 0, 0, jf);
  j[5] := 0;
  j[6] := SEL(t[6] > 0, 0, -jf); 
END_IF

vUppLim := SEL(vMax > 0, vMin, vMax) + 1E-12;
vLowLim := SEL(vMax > 0, vMax, vMin) - 1E-12;

direction := SEL(vMax > 0, ProfileDirection.Down, ProfileDirection.Up);
vUppLim := SEL(direction = ProfileDirection.Up, vMin, vMax) + Constants.VelocityEpsilon;
vLowLim := SEL(direction = ProfileDirection.Up, vMax, vMin) - Constants.VelocityEpsilon;
        
FOR i:= 0 TO 6 
DO
  a[i+1] := a[i] + t[i] * j[i];
  v[i+1] := v[i] + t[i] * (a[i] + t[i] * j[i] / 2);
  p[i+1] := p[i] + t[i] * (v[i] + t[i] * (a[i] / 2 + t[i] * j[i] / 6));

  IF limits = ReachedLimits.Acc0Acc1Vel OR_ELSE limits = ReachedLimits.Acc0Acc1 OR_ELSE limits = ReachedLimits.Acc0Vel OR_ELSE limits = ReachedLimits.Acc1Vel OR_ELSE limits = ReachedLimits.Vel
  THEN
    IF i = 2
    THEN
     a[3] := 0.0;
    END_IF
  END_IF
  
  IF setLimits
  THEN
    IF limits = ReachedLimits.Acc1
    THEN
      IF i = 2
      THEN
        a[3] := aMin;
      END_IF
    ELSIF limits = ReachedLimits.Acc0Acc1
    THEN
      CASE i
      OF
      0: a[1] := aMax;
      4: a[5] := aMin;
      END_CASE  
    END_IF
  END_IF
  
  IF (i > 1 AND_THEN a[i+1] * a[i] < -Constants.DoubleEpsilon) 
  THEN
    v_a_zero := v[i] - (a[i] * a[i]) / (2 * j[i]);
    IF (v_a_zero > vUppLim OR_ELSE v_a_zero < vLowLim)
    THEN
      RETURN;        
		END_IF
  END_IF
END_FOR


THIS^.ControlSigns := controlSigns;
THIS^.Limits := limits;

aUppLim := SEL(direction = ProfileDirection.Up, aMin, aMax) + Constants.AccelerationEpsilon;
aLowLim := SEL(direction = ProfileDirection.Up, aMax, aMin) - Constants.AccelerationEpsilon;

// Velocity limit can be broken in the beginning if both initial velocity and acceleration are too high
CheckVel := ABS(p[7] - pf) < Constants.PositionPrecision
    AND_THEN ABS(v[7] - vf) < Constants.VelocityPrecision
    AND_THEN ABS(a[7] - af) < Constants.AccelerationPrecision // This is not really needed, but we want to double check
    // AND_THEN ABS(v[3]) <= vMaxAbs AND_THEN ABS(v[4]) <= vMaxAbs AND_THEN ABS(v[5]) <= vMaxAbs AND_THEN ABS(v[6]) <= vMaxAbs
    AND_THEN a[1] >= aLowLim AND_THEN a[3] >= aLowLim AND_THEN a[5] >= aLowLim
    AND_THEN a[1] <= aUppLim AND_THEN a[3] <= aUppLim AND_THEN a[5] <= aUppLim
    AND_THEN v[3] <= vUppLim AND_THEN v[4] <= vUppLim AND_THEN v[5] <= vUppLim AND_THEN v[6] <= vUppLim
    AND_THEN v[3] >= vLowLim AND_THEN v[4] >= vLowLim AND_THEN v[5] >= vLowLim AND_THEN v[6] >= vLowLim; // this is not really needed, but we want to double check
END_METHOD

METHOD CheckWithTiming : BOOL
VAR_INPUT
  controlSigns : ProfileControlSigns;    
  limits : ReachedLimits;
  tf : LREAL;
  jf : LREAL;
  vMax : LREAL;
  vMin : LREAL;  
  aMax : LREAL;
  aMin : LREAL;  
END_VAR
// Time doesn't need to be checked as every Profile has a: tf - ... equation
CheckWithTiming := CheckVel(controlSigns, limits, jf, vMax, vMin, aMax, aMin, setLimits:=FALSE); // && (std::abs(t_sum[6] - tf) < Constants.TimePrecision)
END_METHOD

METHOD CheckWithTiming2 : BOOL
VAR_INPUT
  controlSigns : ProfileControlSigns;    
  limits : ReachedLimits;
  tf : LREAL;
  jf : LREAL;
  vMax : LREAL;
  vMin : LREAL;  
  aMax : LREAL;
  aMin : LREAL;
  jMax  : LREAL;
END_VAR
CheckWithTiming2 := (ABS(jf) < ABS(jMax) + Constants.JerkEpsilon) AND_THEN CheckWithTiming(controlSigns, limits, tf, jf, vMax, vMin, aMax, aMin);
END_METHOD

METHOD FirstStateAtPosition : BOOL
VAR_INPUT
  pt, offset : LREAL;
END_VAR
VAR_IN_OUT
  t_t, v_t, a_t : LREAL;
END_VAR
VAR
  i,h : INT;
  p_t : LREAL;
  polynom : ARRAY[0..4] OF LREAL;
  rootCount : INT;
  root : ARRAY[0..6] OF LREAL;
END_VAR
FOR i:=0 TO 6
DO
  IF ABS(p[i] - pt) < Constants.DoubleEpsilon
  THEN
    t_t := offset + SEL(i>0, 0, t_sum[i-1]);
    v_t := v[i];
    a_t := a[i];
    FirstStateAtPosition := TRUE;
    RETURN;
	END_IF
  
  IF t[i] = 0
  THEN
    CONTINUE;
	END_IF
  
  polynom[0] := j[i]/6;
  polynom[1] := a[i]*0.5;
  polynom[2] := v[i];
  polynom[3] := p[i]-pt;
  Roots.SolveCub(ADR(polynom), rootCount:=rootCount, roots:=root);
  FOR h:=0 TO rootCount
  DO
    IF(0 < root[h] AND_THEN root[h] <= t[i])
    THEN
      t_t := offset + root[h] + SEL(i>0, 0, t_sum[i-1]);
      Integrate(root[h], p[i], v[i], a[i], j[i], p_t, v_t, a_t);
      FirstStateAtPosition := TRUE;
      RETURN;      
		END_IF
  END_FOR
  
END_FOR

IF ABS(pf-pt) < Constants.Epsilon
THEN
  t_t := offset + t_sum[6];
  v_t := vf;
  a_t := af;
  FirstStateAtPosition := TRUE;
  RETURN;      
END_IF
END_METHOD

/// Set boundary values for the position interface
METHOD SetBoundary
VAR_IN_OUT CONSTANT
  profile : ProfileDesc;
END_VAR
a[0] := profile.a[0];
v[0] := profile.v[0];
p[0] := profile.p[0];
af := profile.af;
vf := profile.vf;
pf := profile.pf;
Brake := profile.Brake;
Accel := profile.Accel;
END_METHOD

/// Set boundary values for the position interface
METHOD SetBoundaryPosition
VAR_INPUT
  p0_new, v0_new, a0_new, pf_new, vf_new, af_new : LREAL;
END_VAR
a[0] := a0_new;
v[0] := v0_new;
p[0] := p0_new;
af := af_new;
vf := vf_new;
pf := pf_new;
END_METHOD

/// Set boundary values for the velocity interface
METHOD SetBoundaryVelocity
VAR_INPUT
  p0_new, v0_new, a0_new, vf_new, af_new : LREAL;
END_VAR
a[0] := a0_new;
v[0] := v0_new;
p[0] := p0_new;
af := af_new;
vf := vf_new;
END_METHOD

END_FUNCTION_BLOCK

// ---- Struckig/BrakeProfile/BrakeProfile.TcPOU
// Struckig
// Copyright (C) 2022 Stefan Besler

// This program is free software: you can redistribute it and/or modify
// it under the terms of the GNU General Public License as published by
// the Free Software Foundation, either version 3 of the License, or
// (at your option) any later version.

// This program is distributed in the hope that it will be useful,
// but WITHOUT ANY WARRANTY; without even the implied warranty of
// MERCHANTABILITY or FITNESS FOR A PARTICULAR PURPOSE.  See the
// GNU General Public License for more details.
//
// You should have received a copy of the GNU General Public License
// along with THIS PROGRAM.  IF NOT, see <http://www.gnu.org/licenses/>.
/// Calculates (pre- or post-) profile to get current or final state below the limits
FUNCTION_BLOCK BrakeProfile
VAR_INPUT
  Duration : LREAL; //! Overall duration
  t, j, a, v, p : ARRAY[0..2] OF LREAL; //! Profile information for up to three-step profile  
  IsUsed : BOOL;
END_VAR
VAR
  t_to_a_min, t_to_a_max, t_min_to_v_max, t_to_a_zero, t_to_v_min, t_to_v_max : LREAL;
  t_to_v_max_with_constant, t_to_v_min_with_constant, v_at_a0, v_at_a_max, v_at_a_min : LREAL;
END_VAR

METHOD AccelerationBrake
VAR_INPUT
  v0, a0 : LREAL;
  vMax, vMin : LREAL;
  aMax, aMin : LREAL;
  jMax : LREAL;
END_VAR
j[0] := -jMax;

t_to_a_max := (a0 - aMax) / jMax;
t_to_a_zero := a0 / jMax;

v_at_a_max := VelocityAtTime(v0, a0, -jMax, t_to_a_max);
v_at_a0 := VelocityAtTime(v0, a0, -jMax, t_to_a_zero);

IF (v_at_a0 > vMax AND_THEN jMax > 0) OR_ELSE (v_at_a0 < vMax AND_THEN jMax < 0)
THEN
  VelocityBrake(v0, a0, vMax, vMin, aMax, aMin, jMax);

ELSIF (v_at_a_max < vMin AND_THEN jMax > 0) OR_ELSE (v_at_a_max > vMin AND_THEN jMax < 0)
THEN
  t_to_v_min := -(v_at_a_max - vMin)/aMax;
  t_to_v_max := -aMax/(2*jMax) - (v_at_a_max + vMax)/aMax;
  t[0] := t_to_a_max + Constants.BrakeEpsilon;
  t[1] := MAX(MIN(t_to_v_min, v_at_a_max - Constants.BrakeEpsilon), 0.0);
ELSE
  t[0] := t_to_a_max + Constants.BrakeEpsilon;
END_IF
END_METHOD

/// Finalize third-order braking by integrating along kinematic state
METHOD Finalize
VAR_IN_OUT
  ps : LREAL;
  vs : LREAL;
  as : LREAL;
END_VAR
IF t[0] <= 0 AND_THEN t[1] <= 0
THEN
  Duration := 0;
  RETURN;
END_IF

Duration := t[0];
p[0] := ps;
v[0] := vs;
a[0] := as;
Integrate(t[0], p0:=ps, v0:=vs, a0:=as, j:=j[0], p:=ps, v:=vs, a:=as);

IF t[1] > 0
THEN
  Duration := Duration + t[1];
  p[1] := ps;
  v[1] := vs;
  a[1] := as;
  Integrate(t[1], p0:=ps, v0:=vs, a0:=as, j:=j[1], p:=ps, v:=vs, a:=as);
END_IF

IF t[2] > 0
THEN
  Duration := Duration + t[2];
  p[2] := ps;
  v[2] := vs;
  a[2] := as;
  Integrate(t[2], p0:=ps, v0:=vs, a0:=as, j:=j[2], p:=ps, v:=vs, a:=as);
END_IF
END_METHOD

/// Finalize third-order braking by integrating along kinematic state
METHOD FinalizeSecondOrder
VAR_IN_OUT
  ps : LREAL;
  vs : LREAL;
  as : LREAL;
END_VAR
IF t[0] <= 0.0
THEN
  Duration := 0;
  RETURN;
END_IF

Duration := t[0];
p[0] := ps;
v[0] := vs;
Integrate(t[0], p0:=ps, v0:=vs, a0:=a[0], j:=j[0], p:=ps, v:=vs, a:=as);
END_METHOD

/// Calculate brake trajectory for third-order position interface
METHOD PositionBrakeTrajectory
VAR_INPUT
  v0, a0 : LREAL;
  vMax, vMin : LREAL;
  aMax, aMin : LREAL;
  jMax : LREAL;
  SmoothBrake : BOOL;
END_VAR
t[0] := 0.0;
t[1] := 0.0;
t[2] := 0.0;
j[0] := 0.0;
j[1] := 0.0;
j[2] := 0.0;

IF jMax = 0 OR_ELSE aMax = 0 OR_ELSE aMin = 0
THEN
  RETURN;
ELSIF a0 > aMax
THEN
  AccelerationBrake(v0, a0, vMax, vMin, aMax, aMin, jMax);
ELSIF a0 < aMin
THEN
  AccelerationBrake(v0, a0, vMin, vMax, aMin, aMax, -jMax);
ELSIF SmoothBrake AND_THEN v0 > vMax AND_THEN ABS(a0) < aMax
THEN
  SmoothVelocityBrake(v0, a0, vMax, aMax, jMax);
  IF t[0] <= 0 THEN
    VelocityBrake(v0, a0, vMax, vMin, aMax, aMin, jMax);
  END_IF
ELSIF SmoothBrake AND_THEN v0 < vMin AND_THEN ABS(a0) < aMax
THEN
  SmoothVelocityBrake(v0, a0, vMin, aMax, -jMax);
  IF t[0] <= 0 THEN
    VelocityBrake(v0, a0, vMin, vMax, aMin, aMax, -jMax);
  END_IF
ELSIF ((v0 > vMax AND_THEN VelocityAtZeroAcceleration(v0, a0, -jMax) > vMin) OR_ELSE (a0 > 0 AND_THEN VelocityAtZeroAcceleration(v0, a0, jMax) > vMax))
THEN
  VelocityBrake(v0, a0, vMax, vMin, aMax, aMin, jMax);
ELSIF ((v0 < vMin AND_THEN VelocityAtZeroAcceleration(v0, a0, jMax) < vMax) OR_ELSE (a0 < 0 AND_THEN VelocityAtZeroAcceleration(v0, a0, -jMax) < vMin))
THEN
  VelocityBrake(v0, a0, vMin, vMax, aMin, aMax, -jMax);      
END_IF
END_METHOD

/// Calculate brake trajectory for third-order position interface
METHOD SecondOrderPositionBrakeTrajectory
VAR_INPUT
  v0 : LREAL;
  vMax, vMin : LREAL;
  aMax, aMin : LREAL;
END_VAR
t[0] := 0.0;
t[1] := 0.0;
j[0] := 0.0;
j[1] := 0.0;
a[0] := 0.0;
a[1] := 0.0;

IF aMax = 0.0 OR_ELSE aMin = 0.0
THEN
  RETURN; // Ignore braking for zero-limits 
END_IF

IF v0 > vMax
THEN
  a[0] := aMin;
  t[0] := (vMax - v0)/aMin + Constants.Epsilon;   
ELSIF v0 < vMin
THEN
  a[0] := aMax;
  t[0] := (vMin - v0)/aMax + Constants.Epsilon;
END_IF
END_METHOD

/// Calculate brake trajectory for third-order position interface
METHOD SecondOrderVelocityBrakeTrajectory
VAR_INPUT
END_VAR
t[0] := 0;
t[1] := 0;
j[0] := 0;
j[1] := 0;
END_METHOD

/// Jerk-limited brake from (v0, a0) to (vTarget, a=0).
/// Produces a 2- or 3-phase profile that ends with zero acceleration,
/// so Step1 does not inherit a large residual deceleration.
/// jMax > 0 means braking from above (v0 > vTarget), jMax < 0 means from below.
/// If the profile cannot be computed (e.g. a0 opposes braking too strongly),
/// t[0] remains 0 so the caller can fall back to legacy VelocityBrake.
METHOD SmoothVelocityBrake
VAR_INPUT
  v0, a0 : LREAL;
  vTarget : LREAL;
  aMax : LREAL;
  jMax : LREAL;
END_VAR
VAR
  half_D, t1, t3, a_peak : LREAL;
  v1, dv_phase3, t2, a_clamp : LREAL;
END_VAR
IF (jMax > 0 AND_THEN v0 <= vTarget) OR_ELSE (jMax < 0 AND_THEN v0 >= vTarget) THEN
  RETURN;
END_IF

(* Solve quadratic for 2-phase brake from (v0,a0) to (vTarget,0):
   Phase 1: j = -jMax, duration t1
   Phase 3: j = +jMax, duration t3 = t1 - a0/jMax
   jMax * t1^2 - 2*a0*t1 + (vTarget - v0 + a0^2/(2*jMax)) = 0
   D/4 = a0^2/2 + jMax*(v0 - vTarget) *)
half_D := a0*a0*0.5 + jMax*(v0 - vTarget);
IF half_D < 0 THEN
  RETURN;
END_IF

IF jMax > 0 THEN
  t1 := (a0 + SQRT(half_D)) / jMax;
ELSE
  t1 := (a0 - SQRT(half_D)) / jMax;
END_IF

IF t1 < 0 THEN
  RETURN;
END_IF

t3 := t1 - a0/jMax;
a_peak := a0 - jMax*t1;

IF ABS(a_peak) <= aMax THEN
  j[0] := -jMax;
  t[0] := t1;
  j[1] := jMax;
  t[1] := t3;
  t[2] := 0;
ELSE
  (* 3-phase: clamp peak acceleration at ±aMax *)
  IF jMax > 0 THEN
    a_clamp := -aMax;
  ELSE
    a_clamp := aMax;
  END_IF

  t1 := (a0 - a_clamp) / jMax;
  t3 := -a_clamp / jMax;
  v1 := v0 + a0*t1 - 0.5*jMax*t1*t1;
  dv_phase3 := a_clamp*t3 + 0.5*jMax*t3*t3;
  t2 := (vTarget - v1 - dv_phase3) / a_clamp;

  IF t2 < 0 THEN
    RETURN;
  END_IF

  j[0] := -jMax;
  t[0] := t1;
  j[1] := 0;
  t[1] := t2;
  j[2] := jMax;
  t[2] := t3;
END_IF
END_METHOD

METHOD VelocityAtTime : LREAL
VAR_INPUT
  v0, a0 : LREAL;
  j : LREAL;
  t : LREAL;
END_VAR
VelocityAtTime := v0 + t * (a0 + j * t * 0.5);
END_METHOD

METHOD VelocityAtZeroAcceleration : LREAL
VAR_INPUT
  v0, a0 : LREAL;
  j : LREAL;
END_VAR
VelocityAtZeroAcceleration := v0 + (a0 * a0) / (2 * j);
END_METHOD

METHOD VelocityBrake
VAR_INPUT
  v0, a0 : LREAL;
  vMax, vMin : LREAL;
  aMax, aMin : LREAL;
  jMax : LREAL;
END_VAR
j[0] := -jMax;
t_to_a_min := (a0 - aMin)/jMax;
t_to_v_max := a0*a0 + 2 * jMax * (v0 - vMax);
t_to_v_min := a0*a0 / 2 + jMax * (v0 - vMin);

IF t_to_v_max < 0 OR_ELSE t_to_v_min < 0
THEN
  RETURN;
END_IF

t_to_v_max := a0/jMax + SQRT(t_to_v_max) / ABS(jMax);
t_to_v_min := a0/jMax + SQRT(t_to_v_min) / ABS(jMax);
t_min_to_v_max := MIN(t_to_v_max, t_to_v_min);

IF (t_to_a_min < t_min_to_v_max)
THEN
  v_at_a_min := VelocityAtTime(v0, a0, -jMax, t_to_a_min);
  t_to_v_max_with_constant := -(v_at_a_min - vMax)/aMin;
  t_to_v_min_with_constant := -0.5*aMin/jMax - (v_at_a_min - vMin)/aMin;
  t[0] := MAX(t_to_a_min - Constants.BrakeEpsilon, 0);
  t[1] := MAX(MIN(t_to_v_max_with_constant, t_to_v_min_with_constant), 0.0);
ELSE
  t[0] := MAX(t_min_to_v_max - Constants.BrakeEpsilon, 0);
END_IF
END_METHOD

/// Calculate brake trajectory for third-order velocity interface
METHOD VelocityBrakeTrajectory
VAR_INPUT
  v0, a0 : LREAL;
  aMax, aMin : LREAL;
  jMax : LREAL;
END_VAR
t[0] := 0.0;
t[1] := 0.0;
j[0] := 0.0;
j[1] := 0.0;

IF jMax = 0
THEN
  RETURN; // Ignore braking for zero-limits
ELSIF (a0 > aMax)
THEN
  j[0] := -jMax;
  t[0] := (a0 - aMax)/jMax + Constants.BrakeEpsilon;
ELSIF (a0 < aMin)
THEN
  j[0] := jMax;
  t[0] := -(a0 - aMin)/jMax + Constants.BrakeEpsilon;
END_IF
END_METHOD

END_FUNCTION_BLOCK

// ---- Struckig/Integrate.TcPOU
// Struckig
// Copyright (C) 2022 Stefan Besler

// This program is free software: you can redistribute it and/or modify
// it under the terms of the GNU General Public License as published by
// the Free Software Foundation, either version 3 of the License, or
// (at your option) any later version.

// This program is distributed in the hope that it will be useful,
// but WITHOUT ANY WARRANTY; without even the implied warranty of
// MERCHANTABILITY or FITNESS FOR A PARTICULAR PURPOSE.  See the
// GNU General Public License for more details.
//
// You should have received a copy of the GNU General Public License
// along with THIS PROGRAM.  IF NOT, see <http://www.gnu.org/licenses/>.
/// Integrate with constant jerk for duration t. Returns new position, new velocity, and new acceleration.
FUNCTION INTERNAL Integrate
VAR_INPUT
  t, p0, v0, a0, j : LREAL;
END_VAR
VAR_IN_OUT
  p, v, a : LREAL;
END_VAR

p := p0 + t * (v0 + t * (a0 * 0.5 + t * j / 6));
v := v0 + t * (a0 + t * j * 0.5);
a := a0 + t * j;

END_FUNCTION

// ---- Struckig/Math/Roots.TcPOU
// Struckig
// Copyright (C) 2022 Stefan Besler

// This program is free software: you can redistribute it and/or modify
// it under the terms of the GNU General Public License as published by
// the Free Software Foundation, either version 3 of the License, or
// (at your option) any later version.

// This program is distributed in the hope that it will be useful,
// but WITHOUT ANY WARRANTY; without even the implied warranty of
// MERCHANTABILITY or FITNESS FOR A PARTICULAR PURPOSE.  See the
// GNU General Public License for more details.
//
// You should have received a copy of the GNU General Public License
// along with THIS PROGRAM.  IF NOT, see <http://www.gnu.org/licenses/>.
PROGRAM INTERNAL Roots
VAR
  a2, q, qsqrt, r2, q3, aa, t : LREAL;
  a, b, c, d, rr, theta, ux, uyi, inva, invaa, bb, bover3a, p, halfq, yy, inv2b, x, y, uuu, vvv, www, w, h : LREAL;
  discriminant : LREAL;
  e0, e1, q1, q2, p1, p2, dd, sqrtD  : LREAL;
  a3, b3, c3 : LREAL;
  x3 : ARRAY[0..2] OF LREAL;
  number_zeroes : INT;  
  deriv : ARRAY[0 .. 10] OF LREAL;
  fl, fh, temp : LREAL;
  dxold, dx, f,df : LREAL;
  j : INT;
  xn : LREAL;
  iterations : BYTE;
END_VAR

METHOD PolyDeri
VAR_INPUT
  coeffs : POINTER TO LREAL;
  coeffsCount : BYTE;
  out : POINTER TO LREAL;
END_VAR
FOR j:=0 TO coeffsCount DO
  out[j] := (coeffsCount - j) * coeffs[j];
END_FOR
END_METHOD

METHOD PolyEval : LREAL;
VAR_INPUT
  polynom : POINTER TO LREAL;
  degree : INT;
  x : LREAL;
END_VAR
IF degree = 0
THEN
  RETURN;
END_IF

IF (ABS(x) < Constants.DoubleEpsilon) THEN
    PolyEval := polynom[degree];
ELSIF x = 1.0 THEN
  FOR j:= degree TO 0 BY -1
  DO
    PolyEval := PolyEval + polynom[j];
  END_FOR
ELSE
  xn := 1.0;
  FOR j:= degree TO 0 BY -1 
  DO
    PolyEval := PolyEval + polynom[j] * xn;
    xn := xn * x;
  END_FOR
END_IF
END_METHOD

METHOD PolyMonicDeri
VAR_INPUT
  monic_coeffs : POINTER TO LREAL;
  coeffsCount : BYTE;
  out : POINTER TO LREAL;  
END_VAR
VAR
  i : BYTE;
END_VAR
out[0] := 1.0;
FOR i:=1 TO coeffsCount-1 DO
  out[i] := (coeffsCount- i) * (monic_coeffs[i] / (coeffsCount));
END_FOR
END_METHOD

// Calculate a single zero of polynom p(x) inside [lbound, ubound]
// Requirements: p(lbound)*p(ubound) < 0, lbound < ubound
METHOD ShrinkInterval : LREAL
VAR_INPUT
  p : POINTER TO LREAL;
  degree : BYTE;  
  l, h : LREAL;
END_VAR
fl := PolyEval(p, degree, l);
fh := PolyEval(p, degree, h);
IF (fl = 0.0) THEN
  ShrinkInterval := l;
  RETURN;
END_IF

IF (fh = 0.0) THEN
  ShrinkInterval := h;
  RETURN;
END_IF

IF (fl > 0.0)
THEN
  // swap l and h
  temp := l;
  l := h;
  h := temp;
END_IF

ShrinkInterval := (l + h) / 2;
dxold := ABS(h - l);
dx := dxold;
PolyDeri(p, degree, out:=ADR(deriv));
f := PolyEval(p, degree, ShrinkInterval);
df := PolyEval(ADR(deriv), degree-1, ShrinkInterval);
FOR iterations:=0 TO ParameterList.MaxIterations DO
  IF ((((ShrinkInterval - h) * df - f) * ((ShrinkInterval - l) * df - f) > 0.0) OR_ELSE (ABS(2 * f) > ABS(dxold * df))) THEN
    dxold := dx;
    dx := (h - l) / 2;
    ShrinkInterval := l + dx;
    IF (l = ShrinkInterval) THEN
      RETURN;
    END_IF
  ELSE
  
